Yaskawa INFORM job: DEMO_ROOF_SIDE_0625_3PAINT_13.JBI

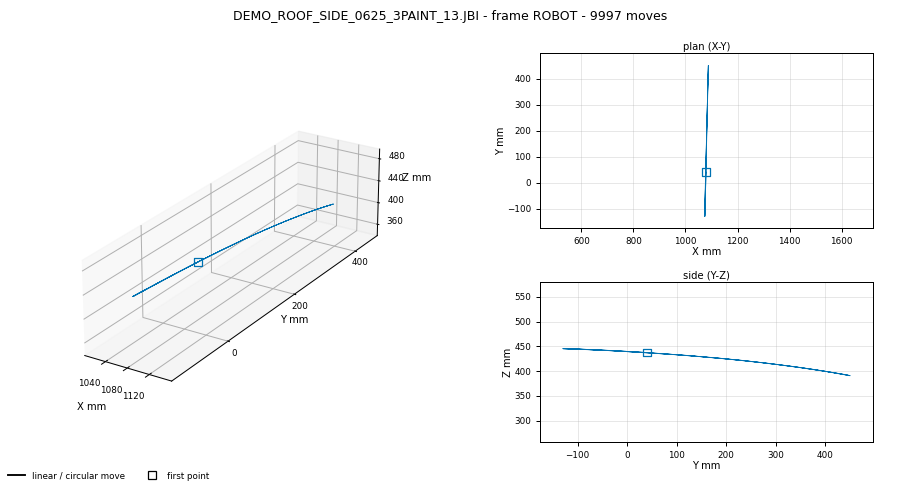
[picture p0: tool path of DEMO_ROOF_SIDE_0625_3PAINT_13.JBI in frame ROBOT, 9997 of 9997 moves have a stored position in this frame; points joined in program order, loops and branches not executed]
/JOB
//NAME DEMO_ROOF_SIDE_0625_3PAINT13
//POS
///NPOS 9997,0,0,0,0,0
///TOOL 0
///USER 0
///POSTYPE ROBOT
///RECTAN
///RCONF 1,0,0,0,0,0,0,0,0,0,0,0,0,0,0,0,0,0,0,0,0,0,0,0
C00000=1079.209,40.966,437.430,173.893,21.647,153.724
C00001=1079.203,40.716,437.445,173.891,21.644,153.724
C00002=1079.197,40.467,437.461,173.890,21.643,153.724
C00003=1079.192,40.217,437.477,173.889,21.640,153.724
C00004=1079.186,39.968,437.493,173.888,21.638,153.723
C00005=1079.181,39.718,437.508,173.885,21.635,153.723
C00006=1079.174,39.469,437.524,173.884,21.633,153.723
C00007=1079.169,39.220,437.539,173.883,21.630,153.723
C00008=1079.163,38.971,437.556,173.881,21.628,153.723
C00009=1079.157,38.721,437.571,173.880,21.625,153.722
C00010=1079.151,38.471,437.587,173.878,21.623,153.722
C00011=1079.145,38.222,437.602,173.877,21.621,153.722
C00012=1079.139,37.973,437.618,173.875,21.618,153.722
C00013=1079.134,37.723,437.634,173.874,21.616,153.721
C00014=1079.129,37.474,437.649,173.873,21.614,153.721
C00015=1079.122,37.225,437.665,173.870,21.611,153.721
C00016=1079.116,36.975,437.680,173.869,21.609,153.721
C00017=1079.111,36.725,437.696,173.868,21.606,153.720
C00018=1079.105,36.476,437.711,173.867,21.605,153.720
C00019=1079.099,36.226,437.726,173.865,21.602,153.720
C00020=1079.093,35.977,437.743,173.863,21.600,153.720
C00021=1079.087,35.727,437.758,173.862,21.597,153.719
C00022=1079.082,35.478,437.773,173.861,21.595,153.719
C00023=1079.076,35.229,437.789,173.859,21.592,153.719
C00024=1079.069,34.979,437.804,173.857,21.590,153.719
C00025=1079.064,34.729,437.820,173.856,21.588,153.719
C00026=1079.058,34.481,437.835,173.855,21.585,153.718
C00027=1079.052,34.231,437.850,173.853,21.583,153.718
C00028=1079.046,33.981,437.866,173.852,21.581,153.718
C00029=1079.041,33.732,437.881,173.850,21.578,153.718
C00030=1079.035,33.483,437.897,173.848,21.576,153.717
C00031=1079.029,33.233,437.912,173.847,21.573,153.717
C00032=1079.023,32.984,437.927,173.846,21.571,153.717
C00033=1079.017,32.734,437.943,173.845,21.569,153.717
C00034=1079.011,32.485,437.958,173.843,21.566,153.716
C00035=1079.006,32.235,437.973,173.841,21.564,153.716
C00036=1079.000,31.985,437.989,173.840,21.562,153.716
C00037=1078.994,31.736,438.004,173.839,21.559,153.716
C00038=1078.988,31.487,438.020,173.837,21.557,153.715
C00039=1078.982,31.206,438.037,173.835,21.554,153.715
C00040=1078.975,30.926,438.054,173.833,21.551,153.715
C00041=1078.969,30.646,438.071,173.832,21.549,153.715
C00042=1078.963,30.365,438.088,173.830,21.546,153.714
C00043=1078.956,30.116,438.104,173.829,21.544,153.714
C00044=1078.951,29.867,438.119,173.828,21.542,153.714
C00045=1078.945,29.617,438.134,173.826,21.539,153.714
C00046=1078.939,29.367,438.150,173.825,21.536,153.713
C00047=1078.933,29.118,438.164,173.823,21.534,153.713
C00048=1078.928,28.868,438.180,173.822,21.532,153.713
C00049=1078.923,28.619,438.195,173.820,21.529,153.713
C00050=1078.916,28.370,438.211,173.819,21.527,153.712
C00051=1078.909,28.120,438.225,173.818,21.524,153.712
C00052=1078.904,27.871,438.241,173.816,21.523,153.712
C00053=1078.898,27.622,438.256,173.814,21.520,153.712
C00054=1078.892,27.372,438.271,173.813,21.517,153.711
C00055=1078.887,27.123,438.286,173.812,21.515,153.711
C00056=1078.881,26.873,438.301,173.810,21.513,153.711
C00057=1078.875,26.624,438.316,173.808,21.510,153.711
C00058=1078.870,26.374,438.331,173.807,21.508,153.711
C00059=1078.863,26.124,438.346,173.806,21.506,153.710
C00060=1078.857,25.875,438.361,173.805,21.503,153.710
C00061=1078.852,25.625,438.376,173.803,21.501,153.710
C00062=1078.846,25.376,438.391,173.801,21.499,153.710
C00063=1078.840,25.126,438.407,173.800,21.496,153.709
C00064=1078.834,24.877,438.421,173.799,21.494,153.709
C00065=1078.828,24.628,438.436,173.798,21.492,153.709
C00066=1078.822,24.378,438.452,173.796,21.489,153.709
C00067=1078.817,24.129,438.466,173.794,21.487,153.708
C00068=1078.810,23.879,438.481,173.793,21.484,153.708
C00069=1078.805,23.630,438.496,173.792,21.482,153.708
C00070=1078.799,23.380,438.511,173.790,21.480,153.708
C00071=1078.794,23.131,438.526,173.789,21.477,153.707
C00072=1078.787,22.881,438.541,173.787,21.475,153.707
C00073=1078.781,22.631,438.556,173.786,21.473,153.707
C00074=1078.776,22.382,438.572,173.784,21.470,153.707
C00075=1078.770,22.133,438.586,173.783,21.468,153.707
C00076=1078.764,21.884,438.601,173.781,21.465,153.706
C00077=1078.758,21.634,438.617,173.780,21.463,153.706
C00078=1078.752,21.385,438.631,173.778,21.460,153.706
C00079=1078.746,21.135,438.646,173.777,21.458,153.706
C00080=1078.741,20.885,438.661,173.776,21.456,153.705
C00081=1078.735,20.635,438.675,173.774,21.454,153.705
C00082=1078.729,20.387,438.690,173.772,21.451,153.705
C00083=1078.724,20.137,438.706,173.771,21.449,153.705
C00084=1078.718,19.888,438.720,173.770,21.447,153.704
C00085=1078.711,19.638,438.735,173.769,21.444,153.704
C00086=1078.706,19.389,438.750,173.767,21.442,153.704
C00087=1078.700,19.138,438.765,173.765,21.439,153.704
C00088=1078.694,18.889,438.779,173.764,21.437,153.703
C00089=1078.688,18.640,438.794,173.763,21.435,153.703
C00090=1078.682,18.391,438.809,173.762,21.432,153.703
C00091=1078.677,18.141,438.824,173.759,21.430,153.703
C00092=1078.671,17.891,438.838,173.758,21.428,153.703
C00093=1078.665,17.642,438.853,173.757,21.425,153.702
C00094=1078.659,17.393,438.868,173.756,21.423,153.702
C00095=1078.653,17.143,438.883,173.754,21.420,153.702
C00096=1078.648,16.894,438.898,173.752,21.418,153.702
C00097=1078.641,16.643,438.912,173.751,21.416,153.701
C00098=1078.636,16.395,438.927,173.750,21.414,153.701
C00099=1078.629,16.145,438.941,173.749,21.411,153.701
C00100=1078.624,15.895,438.955,173.747,21.408,153.701
C00101=1078.618,15.645,438.971,173.745,21.407,153.700
C00102=1078.612,15.396,438.985,173.744,21.404,153.700
C00103=1078.606,15.118,439.002,173.742,21.401,153.700
C00104=1078.599,14.838,439.018,173.741,21.399,153.700
C00105=1078.593,14.560,439.034,173.739,21.396,153.699
C00106=1078.586,14.281,439.051,173.738,21.394,153.699
C00107=1078.581,14.031,439.065,173.737,21.391,153.699
C00108=1078.574,13.781,439.080,173.734,21.389,153.699
C00109=1078.569,13.532,439.095,173.733,21.386,153.698
C00110=1078.562,13.282,439.109,173.732,21.384,153.698
C00111=1078.557,13.033,439.123,173.731,21.382,153.698
C00112=1078.550,12.784,439.138,173.729,21.380,153.698
C00113=1078.545,12.534,439.152,173.727,21.377,153.698
C00114=1078.539,12.285,439.167,173.726,21.375,153.697
C00115=1078.533,12.035,439.181,173.725,21.373,153.697
C00116=1078.527,11.786,439.196,173.723,21.371,153.697
C00117=1078.521,11.536,439.211,173.722,21.368,153.697
C00118=1078.515,11.287,439.224,173.720,21.366,153.696
C00119=1078.509,11.037,439.239,173.719,21.363,153.696
C00120=1078.503,10.787,439.253,173.718,21.361,153.696
C00121=1078.497,10.538,439.268,173.717,21.359,153.696
C00122=1078.491,10.289,439.283,173.714,21.357,153.696
C00123=1078.486,10.039,439.297,173.713,21.354,153.695
C00124=1078.479,9.789,439.312,173.712,21.352,153.695
C00125=1078.474,9.540,439.325,173.711,21.350,153.695
C00126=1078.467,9.291,439.340,173.709,21.348,153.695
C00127=1078.461,9.041,439.354,173.707,21.345,153.694
C00128=1078.456,8.792,439.368,173.706,21.343,153.694
C00129=1078.449,8.542,439.382,173.705,21.340,153.694
C00130=1078.444,8.293,439.397,173.703,21.338,153.694
C00131=1078.438,8.042,439.411,173.702,21.336,153.693
C00132=1078.432,7.794,439.426,173.700,21.333,153.693
C00133=1078.426,7.544,439.440,173.699,21.331,153.693
C00134=1078.420,7.294,439.455,173.698,21.329,153.693
C00135=1078.415,7.045,439.469,173.697,21.327,153.693
C00136=1078.409,6.796,439.483,173.694,21.324,153.692
C00137=1078.403,6.546,439.497,173.693,21.322,153.692
C00138=1078.397,6.296,439.511,173.692,21.319,153.692
C00139=1078.391,6.047,439.526,173.691,21.317,153.692
C00140=1078.385,5.797,439.540,173.690,21.315,153.691
C00141=1078.380,5.548,439.555,173.687,21.312,153.691
C00142=1078.373,5.298,439.568,173.686,21.310,153.691
C00143=1078.367,5.048,439.582,173.685,21.308,153.691
C00144=1078.361,4.799,439.597,173.684,21.305,153.691
C00145=1078.356,4.550,439.611,173.682,21.304,153.690
C00146=1078.350,4.300,439.625,173.680,21.301,153.690
C00147=1078.344,4.050,439.639,173.679,21.299,153.690
C00148=1078.339,3.801,439.653,173.678,21.296,153.690
C00149=1078.332,3.551,439.668,173.677,21.294,153.689
C00150=1078.327,3.302,439.682,173.675,21.292,153.689
C00151=1078.321,3.052,439.696,173.673,21.289,153.689
C00152=1078.314,2.803,439.710,173.672,21.287,153.689
C00153=1078.309,2.553,439.724,173.671,21.284,153.688
C00154=1078.303,2.304,439.738,173.670,21.282,153.688
C00155=1078.297,2.055,439.753,173.668,21.280,153.688
C00156=1078.291,1.804,439.767,173.666,21.277,153.688
C00157=1078.286,1.555,439.781,173.665,21.275,153.688
C00158=1078.280,1.305,439.795,173.664,21.273,153.687
C00159=1078.275,1.056,439.809,173.663,21.271,153.687
C00160=1078.268,0.806,439.823,173.661,21.269,153.687
C00161=1078.262,0.557,439.837,173.659,21.266,153.687
C00162=1078.257,0.308,439.851,173.658,21.264,153.687
C00163=1078.251,0.058,439.865,173.657,21.261,153.686
C00164=1078.245,-0.192,439.879,173.655,21.259,153.686
C00165=1078.240,-0.442,439.893,173.654,21.257,153.686
C00166=1078.233,-0.691,439.906,173.652,21.254,153.686
C00167=1078.227,-0.968,439.923,173.651,21.252,153.685
C00168=1078.221,-1.244,439.938,173.649,21.249,153.685
C00169=1078.214,-1.522,439.953,173.648,21.246,153.685
C00170=1078.207,-1.799,439.969,173.647,21.244,153.684
C00171=1078.202,-2.048,439.983,173.644,21.242,153.684
C00172=1078.196,-2.298,439.997,173.643,21.239,153.684
C00173=1078.191,-2.547,440.011,173.642,21.237,153.684
C00174=1078.185,-2.797,440.024,173.641,21.235,153.684
C00175=1078.178,-3.046,440.039,173.640,21.233,153.683
C00176=1078.173,-3.296,440.053,173.638,21.230,153.683
C00177=1078.167,-3.545,440.067,173.636,21.228,153.683
C00178=1078.161,-3.795,440.080,173.635,21.225,153.683
C00179=1078.156,-4.044,440.094,173.634,21.223,153.683
C00180=1078.149,-4.294,440.108,173.632,21.221,153.682
C00181=1078.143,-4.544,440.122,173.630,21.218,153.682
C00182=1078.138,-4.793,440.135,173.629,21.217,153.682
C00183=1078.132,-5.043,440.149,173.628,21.214,153.682
C00184=1078.125,-5.292,440.164,173.627,21.212,153.681
C00185=1078.119,-5.542,440.177,173.625,21.210,153.681
C00186=1078.114,-5.791,440.191,173.624,21.208,153.681
C00187=1078.108,-6.041,440.205,173.622,21.205,153.681
C00188=1078.101,-6.291,440.218,173.621,21.203,153.681
C00189=1078.096,-6.540,440.232,173.619,21.201,153.680
C00190=1078.090,-6.789,440.245,173.618,21.199,153.680
C00191=1078.084,-7.039,440.259,173.617,21.196,153.680
C00192=1078.078,-7.288,440.273,173.615,21.194,153.680
C00193=1078.072,-7.539,440.287,173.614,21.191,153.680
C00194=1078.066,-7.788,440.300,173.612,21.189,153.679
C00195=1078.060,-8.037,440.314,173.611,21.187,153.679
C00196=1078.055,-8.287,440.328,173.610,21.185,153.679
C00197=1078.049,-8.536,440.341,173.608,21.183,153.679
C00198=1078.043,-8.786,440.355,173.607,21.180,153.679
C00199=1078.036,-9.036,440.369,173.605,21.178,153.678
C00200=1078.031,-9.285,440.382,173.604,21.176,153.678
C00201=1078.025,-9.535,440.396,173.603,21.174,153.678
C00202=1078.019,-9.784,440.409,173.601,21.172,153.678
C00203=1078.013,-10.034,440.423,173.599,21.169,153.677
C00204=1078.007,-10.283,440.437,173.598,21.167,153.677
C00205=1078.001,-10.532,440.450,173.597,21.164,153.677
C00206=1077.995,-10.783,440.463,173.596,21.162,153.677
C00207=1077.989,-11.033,440.477,173.594,21.160,153.677
C00208=1077.984,-11.282,440.491,173.592,21.157,153.676
C00209=1077.977,-11.531,440.504,173.591,21.156,153.676
C00210=1077.972,-11.781,440.518,173.590,21.153,153.676
C00211=1077.966,-12.030,440.531,173.588,21.151,153.676
C00212=1077.960,-12.280,440.545,173.587,21.149,153.676
C00213=1077.954,-12.529,440.558,173.586,21.147,153.675
C00214=1077.949,-12.779,440.572,173.584,21.144,153.675
C00215=1077.943,-13.028,440.585,173.582,21.142,153.675
C00216=1077.937,-13.279,440.599,173.581,21.140,153.675
C00217=1077.930,-13.528,440.612,173.580,21.138,153.675
C00218=1077.925,-13.778,440.626,173.579,21.135,153.674
C00219=1077.919,-14.027,440.639,173.578,21.133,153.674
C00220=1077.913,-14.276,440.653,173.575,21.131,153.674
C00221=1077.907,-14.526,440.666,173.574,21.128,153.674
C00222=1077.902,-14.776,440.679,173.573,21.126,153.674
C00223=1077.896,-15.025,440.693,173.572,21.124,153.673
C00224=1077.890,-15.275,440.707,173.570,21.122,153.673
C00225=1077.884,-15.525,440.719,173.568,21.120,153.673
C00226=1077.878,-15.774,440.732,173.567,21.117,153.673
C00227=1077.873,-16.023,440.746,173.566,21.115,153.672
C00228=1077.866,-16.273,440.760,173.564,21.113,153.672
C00229=1077.860,-16.523,440.773,173.563,21.111,153.672
C00230=1077.854,-16.773,440.786,173.562,21.109,153.672
C00231=1077.847,-17.048,440.801,173.560,21.106,153.672
C00232=1077.841,-17.323,440.815,173.559,21.104,153.671
C00233=1077.835,-17.598,440.830,173.556,21.101,153.671
C00234=1077.827,-17.874,440.844,173.555,21.099,153.671
C00235=1077.822,-18.123,440.858,173.554,21.097,153.671
C00236=1077.816,-18.373,440.871,173.553,21.095,153.671
C00237=1077.810,-18.622,440.884,173.552,21.092,153.670
C00238=1077.804,-18.872,440.898,173.549,21.090,153.670
C00239=1077.798,-19.121,440.911,173.548,21.088,153.670
C00240=1077.792,-19.371,440.924,173.547,21.086,153.670
C00241=1077.786,-19.620,440.937,173.546,21.084,153.670
C00242=1077.780,-19.870,440.951,173.544,21.082,153.670
C00243=1077.775,-20.120,440.963,173.543,21.080,153.669
C00244=1077.768,-20.369,440.977,173.541,21.077,153.669
C00245=1077.762,-20.618,440.990,173.540,21.075,153.669
C00246=1077.757,-20.869,441.003,173.538,21.073,153.669
C00247=1077.751,-21.118,441.016,173.537,21.071,153.669
C00248=1077.745,-21.368,441.029,173.536,21.068,153.668
C00249=1077.739,-21.617,441.042,173.534,21.066,153.668
C00250=1077.733,-21.867,441.056,173.532,21.064,153.668
C00251=1077.727,-22.116,441.068,173.531,21.062,153.668
C00252=1077.721,-22.366,441.082,173.530,21.060,153.668
C00253=1077.715,-22.616,441.094,173.529,21.058,153.667
C00254=1077.710,-22.865,441.108,173.527,21.056,153.667
C00255=1077.704,-23.115,441.121,173.526,21.053,153.667
C00256=1077.697,-23.364,441.134,173.525,21.051,153.667
C00257=1077.691,-23.614,441.147,173.523,21.049,153.667
C00258=1077.685,-23.864,441.160,173.521,21.047,153.666
C00259=1077.680,-24.113,441.174,173.520,21.044,153.666
C00260=1077.674,-24.363,441.186,173.519,21.042,153.666
C00261=1077.668,-24.612,441.199,173.517,21.040,153.666
C00262=1077.662,-24.862,441.212,173.516,21.038,153.666
C00263=1077.656,-25.111,441.225,173.514,21.035,153.665
C00264=1077.650,-25.362,441.238,173.513,21.033,153.665
C00265=1077.644,-25.611,441.252,173.511,21.031,153.665
C00266=1077.639,-25.860,441.264,173.510,21.029,153.665
C00267=1077.633,-26.110,441.276,173.509,21.027,153.665
C00268=1077.627,-26.359,441.290,173.508,21.025,153.664
C00269=1077.622,-26.609,441.303,173.505,21.023,153.664
C00270=1077.615,-26.859,441.316,173.504,21.021,153.664
C00271=1077.610,-27.109,441.329,173.503,21.018,153.664
C00272=1077.603,-27.358,441.342,173.502,21.016,153.664
C00273=1077.597,-27.608,441.355,173.500,21.014,153.664
C00274=1077.591,-27.858,441.367,173.499,21.012,153.663
C00275=1077.585,-28.107,441.380,173.498,21.010,153.663
C00276=1077.579,-28.357,441.393,173.496,21.008,153.663
C00277=1077.573,-28.606,441.406,173.494,21.006,153.663
C00278=1077.567,-28.856,441.419,173.493,21.003,153.663
C00279=1077.561,-29.106,441.431,173.492,21.001,153.663
C00280=1077.555,-29.355,441.445,173.490,20.999,153.662
C00281=1077.549,-29.605,441.457,173.489,20.997,153.662
C00282=1077.543,-29.854,441.470,173.488,20.996,153.662
C00283=1077.538,-30.103,441.483,173.486,20.993,153.662
C00284=1077.532,-30.353,441.495,173.484,20.991,153.662
C00285=1077.526,-30.602,441.508,173.483,20.989,153.662
C00286=1077.520,-30.852,441.521,173.482,20.987,153.661
C00287=1077.514,-31.102,441.534,173.481,20.985,153.661
C00288=1077.508,-31.351,441.547,173.479,20.983,153.661
C00289=1077.502,-31.601,441.559,173.478,20.981,153.661
C00290=1077.495,-31.851,441.571,173.476,20.978,153.661
C00291=1077.489,-32.101,441.584,173.474,20.976,153.661
C00292=1077.483,-32.349,441.597,173.473,20.974,153.660
C00293=1077.478,-32.599,441.609,173.472,20.972,153.660
C00294=1077.472,-32.849,441.622,173.471,20.970,153.660
C00295=1077.465,-33.124,441.636,173.469,20.968,153.660
C00296=1077.459,-33.398,441.651,173.467,20.966,153.660
C00297=1077.453,-33.673,441.664,173.466,20.964,153.659
C00298=1077.446,-33.948,441.678,173.464,20.961,153.659
C00299=1077.440,-34.197,441.691,173.462,20.959,153.659
C00300=1077.434,-34.446,441.704,173.461,20.957,153.659
C00301=1077.428,-34.696,441.716,173.460,20.955,153.659
C00302=1077.422,-34.945,441.728,173.458,20.953,153.659
C00303=1077.416,-35.195,441.741,173.457,20.951,153.658
C00304=1077.410,-35.445,441.753,173.456,20.949,153.658
C00305=1077.403,-35.694,441.766,173.455,20.947,153.658
C00306=1077.398,-35.944,441.779,173.453,20.944,153.658
C00307=1077.392,-36.194,441.791,173.451,20.942,153.658
C00308=1077.386,-36.443,441.804,173.450,20.940,153.658
C00309=1077.380,-36.693,441.816,173.449,20.938,153.657
C00310=1077.375,-36.943,441.829,173.447,20.936,153.657
C00311=1077.369,-37.192,441.841,173.446,20.934,153.657
C00312=1077.363,-37.442,441.854,173.445,20.932,153.657
C00313=1077.356,-37.691,441.866,173.442,20.930,153.657
C00314=1077.350,-37.941,441.879,173.441,20.928,153.657
C00315=1077.345,-38.190,441.891,173.440,20.926,153.656
C00316=1077.339,-38.440,441.904,173.438,20.924,153.656
C00317=1077.333,-38.690,441.916,173.437,20.922,153.656
C00318=1077.327,-38.940,441.929,173.436,20.920,153.656
C00319=1077.321,-39.190,441.941,173.434,20.918,153.656
C00320=1077.315,-39.439,441.953,173.433,20.916,153.656
C00321=1077.310,-39.689,441.965,173.431,20.913,153.656
C00322=1077.303,-39.938,441.979,173.430,20.911,153.655
C00323=1077.297,-40.187,441.991,173.428,20.909,153.655
C00324=1077.291,-40.437,442.003,173.427,20.907,153.655
C00325=1077.286,-40.686,442.015,173.426,20.906,153.655
C00326=1077.279,-40.936,442.027,173.424,20.904,153.655
C00327=1077.273,-41.186,442.040,173.423,20.902,153.655
C00328=1077.267,-41.436,442.052,173.422,20.900,153.654
C00329=1077.260,-41.685,442.064,173.420,20.897,153.654
C00330=1077.255,-41.935,442.077,173.418,20.895,153.654
C00331=1077.249,-42.184,442.089,173.417,20.893,153.654
C00332=1077.243,-42.434,442.102,173.416,20.891,153.654
C00333=1077.237,-42.684,442.114,173.414,20.889,153.654
C00334=1077.231,-42.933,442.126,173.413,20.887,153.653
C00335=1077.225,-43.183,442.138,173.412,20.885,153.653
C00336=1077.219,-43.433,442.150,173.410,20.883,153.653
C00337=1077.213,-43.682,442.163,173.409,20.882,153.653
C00338=1077.208,-43.932,442.175,173.407,20.879,153.653
C00339=1077.201,-44.182,442.186,173.405,20.878,153.653
C00340=1077.195,-44.432,442.199,173.404,20.876,153.653
C00341=1077.189,-44.682,442.211,173.403,20.874,153.652
C00342=1077.183,-44.930,442.223,173.401,20.872,153.652
C00343=1077.177,-45.180,442.236,173.400,20.870,153.652
C00344=1077.172,-45.430,442.248,173.399,20.868,153.652
C00345=1077.165,-45.679,442.260,173.397,20.866,153.652
C00346=1077.160,-45.929,442.272,173.396,20.864,153.652
C00347=1077.154,-46.179,442.285,173.394,20.861,153.652
C00348=1077.147,-46.428,442.297,173.392,20.859,153.651
C00349=1077.142,-46.678,442.308,173.391,20.858,153.651
C00350=1077.135,-46.928,442.320,173.390,20.856,153.651
C00351=1077.129,-47.178,442.333,173.388,20.854,153.651
C00352=1077.124,-47.427,442.345,173.387,20.852,153.651
C00353=1077.118,-47.676,442.357,173.386,20.850,153.651
C00354=1077.112,-47.926,442.369,173.384,20.848,153.651
C00355=1077.107,-48.176,442.381,173.383,20.846,153.650
C00356=1077.100,-48.426,442.393,173.381,20.844,153.650
C00357=1077.094,-48.676,442.405,173.380,20.842,153.650
C00358=1077.088,-48.924,442.417,173.378,20.840,153.650
C00359=1077.081,-49.200,442.431,173.377,20.838,153.650
C00360=1077.075,-49.474,442.444,173.376,20.836,153.650
C00361=1077.069,-49.749,442.457,173.373,20.833,153.650
C00362=1077.062,-50.024,442.470,173.372,20.831,153.649
C00363=1077.056,-50.273,442.482,173.371,20.829,153.649
C00364=1077.051,-50.524,442.494,173.369,20.828,153.649
C00365=1077.044,-50.773,442.506,173.368,20.826,153.649
C00366=1077.039,-51.023,442.518,173.367,20.824,153.649
C00367=1077.032,-51.272,442.530,173.364,20.821,153.649
C00368=1077.026,-51.522,442.541,173.363,20.820,153.649
C00369=1077.020,-51.772,442.554,173.362,20.818,153.649
C00370=1077.014,-52.021,442.565,173.360,20.816,153.648
C00371=1077.007,-52.271,442.577,173.359,20.815,153.648
C00372=1077.001,-52.521,442.589,173.357,20.813,153.648
C00373=1076.995,-52.770,442.601,173.356,20.811,153.648
C00374=1076.989,-53.020,442.613,173.355,20.809,153.648
C00375=1076.983,-53.270,442.625,173.353,20.807,153.648
C00376=1076.977,-53.519,442.636,173.352,20.805,153.648
C00377=1076.970,-53.768,442.648,173.351,20.803,153.648
C00378=1076.965,-54.019,442.660,173.348,20.801,153.648
C00379=1076.959,-54.268,442.672,173.347,20.799,153.647
C00380=1076.952,-54.517,442.684,173.346,20.798,153.647
C00381=1076.946,-54.768,442.695,173.344,20.796,153.647
C00382=1076.940,-55.017,442.707,173.343,20.794,153.647
C00383=1076.934,-55.266,442.719,173.341,20.792,153.647
C00384=1076.928,-55.517,442.731,173.340,20.791,153.647
C00385=1076.922,-55.766,442.742,173.339,20.789,153.647
C00386=1076.916,-56.016,442.754,173.337,20.787,153.647
C00387=1076.910,-56.265,442.765,173.336,20.785,153.647
C00388=1076.904,-56.515,442.778,173.334,20.783,153.646
C00389=1076.898,-56.765,442.789,173.333,20.781,153.646
C00390=1076.891,-57.014,442.801,173.331,20.779,153.646
C00391=1076.886,-57.264,442.812,173.329,20.777,153.646
C00392=1076.879,-57.514,442.824,173.328,20.776,153.646
C00393=1076.873,-57.763,442.835,173.327,20.774,153.646
C00394=1076.867,-58.013,442.847,173.325,20.772,153.646
C00395=1076.862,-58.263,442.859,173.324,20.771,153.646
C00396=1076.855,-58.512,442.871,173.322,20.769,153.646
C00397=1076.849,-58.762,442.882,173.321,20.767,153.645
C00398=1076.843,-59.011,442.893,173.320,20.765,153.645
C00399=1076.837,-59.261,442.906,173.318,20.763,153.645
C00400=1076.831,-59.511,442.917,173.317,20.761,153.645
C00401=1076.825,-59.761,442.928,173.315,20.760,153.645
C00402=1076.819,-60.010,442.940,173.314,20.758,153.645
C00403=1076.813,-60.260,442.952,173.312,20.756,153.645
C00404=1076.807,-60.509,442.963,173.310,20.754,153.645
C00405=1076.801,-60.759,442.974,173.309,20.752,153.645
C00406=1076.795,-61.009,442.987,173.308,20.751,153.645
C00407=1076.789,-61.259,442.998,173.306,20.749,153.644
C00408=1076.782,-61.508,443.010,173.305,20.747,153.644
C00409=1076.777,-61.758,443.021,173.303,20.745,153.644
C00410=1076.770,-62.007,443.033,173.302,20.743,153.644
C00411=1076.765,-62.257,443.044,173.301,20.742,153.644
C00412=1076.759,-62.507,443.055,173.299,20.740,153.644
C00413=1076.753,-62.756,443.067,173.298,20.738,153.644
C00414=1076.746,-63.006,443.078,173.296,20.736,153.644
C00415=1076.741,-63.256,443.090,173.295,20.735,153.644
C00416=1076.735,-63.506,443.102,173.294,20.733,153.643
C00417=1076.729,-63.755,443.113,173.292,20.731,153.643
C00418=1076.722,-64.005,443.124,173.290,20.729,153.643
C00419=1076.717,-64.254,443.135,173.289,20.727,153.643
C00420=1076.711,-64.504,443.148,173.287,20.726,153.643
C00421=1076.705,-64.754,443.159,173.286,20.724,153.643
C00422=1076.699,-65.003,443.170,173.284,20.722,153.643
C00423=1076.692,-65.280,443.183,173.283,20.720,153.643
C00424=1076.686,-65.556,443.196,173.282,20.718,153.643
C00425=1076.678,-65.831,443.208,173.279,20.716,153.643
C00426=1076.672,-66.108,443.220,173.278,20.714,153.643
C00427=1076.666,-66.357,443.232,173.277,20.712,153.642
C00428=1076.661,-66.607,443.243,173.275,20.711,153.642
C00429=1076.655,-66.857,443.254,173.274,20.709,153.642
C00430=1076.649,-67.107,443.266,173.272,20.708,153.642
C00431=1076.643,-67.356,443.277,173.271,20.706,153.642
C00432=1076.636,-67.606,443.288,173.269,20.704,153.642
C00433=1076.630,-67.856,443.299,173.268,20.702,153.642
C00434=1076.625,-68.105,443.312,173.266,20.701,153.642
C00435=1076.619,-68.355,443.323,173.265,20.699,153.642
C00436=1076.613,-68.605,443.334,173.264,20.697,153.642
C00437=1076.607,-68.855,443.345,173.262,20.695,153.641
C00438=1076.601,-69.104,443.356,173.260,20.693,153.641
C00439=1076.595,-69.353,443.367,173.259,20.691,153.641
C00440=1076.589,-69.603,443.379,173.257,20.690,153.641
C00441=1076.584,-69.853,443.390,173.256,20.688,153.641
C00442=1076.577,-70.103,443.401,173.254,20.687,153.641
C00443=1076.571,-70.352,443.413,173.253,20.685,153.641
C00444=1076.566,-70.602,443.424,173.251,20.683,153.641
C00445=1076.559,-70.852,443.435,173.250,20.682,153.641
C00446=1076.553,-71.101,443.446,173.249,20.680,153.641
C00447=1076.548,-71.351,443.457,173.247,20.678,153.641
C00448=1076.542,-71.601,443.469,173.246,20.676,153.641
C00449=1076.536,-71.850,443.480,173.244,20.675,153.641
C00450=1076.530,-72.100,443.491,173.243,20.673,153.640
C00451=1076.524,-72.350,443.502,173.241,20.671,153.640
C00452=1076.518,-72.599,443.513,173.240,20.669,153.640
C00453=1076.512,-72.849,443.524,173.239,20.668,153.640
C00454=1076.506,-73.099,443.535,173.237,20.666,153.640
C00455=1076.500,-73.349,443.546,173.236,20.665,153.640
C00456=1076.495,-73.598,443.557,173.234,20.663,153.640
C00457=1076.488,-73.848,443.568,173.233,20.661,153.640
C00458=1076.483,-74.097,443.581,173.231,20.660,153.640
C00459=1076.477,-74.347,443.591,173.230,20.658,153.640
C00460=1076.470,-74.597,443.602,173.229,20.656,153.640
C00461=1076.464,-74.846,443.613,173.227,20.655,153.640
C00462=1076.458,-75.096,443.624,173.226,20.653,153.640
C00463=1076.452,-75.346,443.635,173.223,20.651,153.639
C00464=1076.447,-75.595,443.646,173.222,20.649,153.639
C00465=1076.440,-75.846,443.657,173.220,20.648,153.639
C00466=1076.435,-76.095,443.668,173.219,20.647,153.639
C00467=1076.429,-76.345,443.679,173.217,20.645,153.639
C00468=1076.422,-76.595,443.690,173.216,20.643,153.639
C00469=1076.416,-76.844,443.700,173.214,20.642,153.639
C00470=1076.410,-77.093,443.711,173.213,20.640,153.639
C00471=1076.404,-77.344,443.723,173.212,20.638,153.639
C00472=1076.398,-77.593,443.733,173.210,20.637,153.639
C00473=1076.392,-77.843,443.744,173.209,20.635,153.639
C00474=1076.386,-78.093,443.756,173.207,20.633,153.639
C00475=1076.380,-78.342,443.766,173.206,20.632,153.639
C00476=1076.375,-78.592,443.777,173.204,20.630,153.639
C00477=1076.368,-78.842,443.788,173.203,20.629,153.639
C00478=1076.362,-79.091,443.799,173.201,20.628,153.639
C00479=1076.356,-79.341,443.810,173.200,20.626,153.639
C00480=1076.350,-79.590,443.821,173.198,20.624,153.639
C00481=1076.344,-79.840,443.832,173.197,20.623,153.639
C00482=1076.338,-80.090,443.843,173.195,20.621,153.638
C00483=1076.332,-80.339,443.853,173.194,20.620,153.638
C00484=1076.325,-80.589,443.864,173.192,20.618,153.638
C00485=1076.320,-80.839,443.874,173.191,20.616,153.638
C00486=1076.313,-81.089,443.885,173.189,20.615,153.638
C00487=1076.306,-81.367,443.897,173.188,20.614,153.638
C00488=1076.299,-81.646,443.909,173.186,20.612,153.638
C00489=1076.293,-81.924,443.921,173.184,20.610,153.638
C00490=1076.286,-82.202,443.933,173.183,20.608,153.638
C00491=1076.280,-82.452,443.944,173.181,20.607,153.638
C00492=1076.273,-82.702,443.954,173.180,20.605,153.638
C00493=1076.267,-82.951,443.965,173.178,20.604,153.638
C00494=1076.262,-83.201,443.976,173.177,20.602,153.638
C00495=1076.255,-83.450,443.986,173.175,20.601,153.638
C00496=1076.249,-83.701,443.997,173.173,20.600,153.638
C00497=1076.243,-83.950,444.008,173.172,20.598,153.638
C00498=1076.237,-84.199,444.018,173.170,20.597,153.638
C00499=1076.231,-84.450,444.029,173.169,20.595,153.638
C00500=1076.225,-84.699,444.040,173.167,20.594,153.638
C00501=1076.219,-84.949,444.050,173.166,20.592,153.638
C00502=1076.213,-85.198,444.061,173.164,20.591,153.638
C00503=1076.207,-85.449,444.072,173.163,20.589,153.638
C00504=1076.200,-85.698,444.082,173.161,20.588,153.638
C00505=1076.194,-85.947,444.093,173.160,20.587,153.638
C00506=1076.189,-86.197,444.103,173.158,20.585,153.638
C00507=1076.182,-86.447,444.114,173.157,20.584,153.638
C00508=1076.176,-86.697,444.125,173.155,20.582,153.638
C00509=1076.170,-86.946,444.135,173.154,20.581,153.638
C00510=1076.164,-87.196,444.145,173.152,20.579,153.638
C00511=1076.158,-87.446,444.156,173.151,20.578,153.638
C00512=1076.151,-87.695,444.167,173.149,20.576,153.638
C00513=1076.146,-87.945,444.178,173.148,20.575,153.638
C00514=1076.140,-88.195,444.187,173.146,20.574,153.638
C00515=1076.133,-88.445,444.198,173.145,20.572,153.638
C00516=1076.127,-88.694,444.209,173.143,20.571,153.638
C00517=1076.121,-88.944,444.219,173.141,20.569,153.638
C00518=1076.116,-89.194,444.230,173.140,20.568,153.637
C00519=1076.109,-89.443,444.240,173.138,20.566,153.637
C00520=1076.103,-89.694,444.251,173.137,20.565,153.637
C00521=1076.097,-89.943,444.261,173.135,20.563,153.637
C00522=1076.091,-90.192,444.272,173.134,20.562,153.637
C00523=1076.085,-90.442,444.282,173.132,20.561,153.637
C00524=1076.079,-90.692,444.292,173.131,20.559,153.637
C00525=1076.073,-90.941,444.303,173.129,20.558,153.637
C00526=1076.067,-91.192,444.314,173.129,20.557,153.637
C00527=1076.061,-91.441,444.324,173.127,20.555,153.637
C00528=1076.055,-91.691,444.334,173.126,20.554,153.637
C00529=1076.049,-91.940,444.344,173.124,20.553,153.637
C00530=1076.043,-92.190,444.355,173.122,20.551,153.637
C00531=1076.037,-92.440,444.365,173.121,20.550,153.637
C00532=1076.031,-92.689,444.376,173.119,20.548,153.637
C00533=1076.024,-92.940,444.386,173.118,20.547,153.637
C00534=1076.019,-93.189,444.396,173.116,20.546,153.637
C00535=1076.013,-93.439,444.407,173.115,20.544,153.637
C00536=1076.007,-93.688,444.417,173.113,20.543,153.637
C00537=1076.001,-93.938,444.428,173.112,20.541,153.637
C00538=1075.995,-94.188,444.437,173.110,20.540,153.637
C00539=1075.989,-94.437,444.448,173.108,20.539,153.637
C00540=1075.983,-94.687,444.458,173.107,20.537,153.637
C00541=1075.976,-94.937,444.469,173.105,20.536,153.637
C00542=1075.970,-95.187,444.479,173.104,20.535,153.637
C00543=1075.965,-95.436,444.489,173.102,20.533,153.637
C00544=1075.958,-95.686,444.499,173.101,20.532,153.637
C00545=1075.953,-95.936,444.510,173.099,20.531,153.637
C00546=1075.946,-96.186,444.519,173.098,20.529,153.637
C00547=1075.941,-96.435,444.530,173.096,20.528,153.637
C00548=1075.935,-96.685,444.540,173.095,20.526,153.637
C00549=1075.929,-96.934,444.551,173.093,20.525,153.637
C00550=1075.923,-97.184,444.560,173.091,20.524,153.637
C00551=1075.916,-97.465,444.572,173.090,20.522,153.637
C00552=1075.909,-97.746,444.583,173.088,20.521,153.637
C00553=1075.903,-98.026,444.595,173.087,20.520,153.637
C00554=1075.896,-98.307,444.607,173.085,20.518,153.637
C00555=1075.890,-98.556,444.616,173.084,20.517,153.637
C00556=1075.882,-98.806,444.627,173.082,20.516,153.637
C00557=1075.877,-99.056,444.637,173.080,20.514,153.637
C00558=1075.871,-99.306,444.647,173.079,20.513,153.637
C00559=1075.864,-99.555,444.657,173.077,20.512,153.637
C00560=1075.859,-99.805,444.667,173.076,20.511,153.637
C00561=1075.852,-100.055,444.677,173.074,20.509,153.637
C00562=1075.846,-100.304,444.687,173.072,20.508,153.637
C00563=1075.841,-100.555,444.697,173.071,20.507,153.637
C00564=1075.834,-100.804,444.707,173.069,20.505,153.637
C00565=1075.828,-101.054,444.717,173.068,20.505,153.638
C00566=1075.822,-101.303,444.728,173.066,20.503,153.638
C00567=1075.816,-101.554,444.738,173.065,20.502,153.638
C00568=1075.810,-101.803,444.747,173.063,20.501,153.638
C00569=1075.803,-102.052,444.757,173.062,20.500,153.638
C00570=1075.798,-102.303,444.768,173.060,20.499,153.638
C00571=1075.791,-102.552,444.777,173.059,20.497,153.638
C00572=1075.785,-102.802,444.787,173.057,20.496,153.638
C00573=1075.780,-103.052,444.798,173.056,20.495,153.638
C00574=1075.773,-103.301,444.807,173.054,20.494,153.638
C00575=1075.767,-103.551,444.817,173.053,20.492,153.638
C00576=1075.761,-103.800,444.827,173.051,20.491,153.638
C00577=1075.755,-104.051,444.837,173.049,20.490,153.638
C00578=1075.749,-104.300,444.847,173.048,20.489,153.638
C00579=1075.743,-104.550,444.857,173.046,20.487,153.638
C00580=1075.736,-104.799,444.867,173.044,20.487,153.638
C00581=1075.731,-105.049,444.877,173.043,20.485,153.638
C00582=1075.725,-105.299,444.886,173.041,20.484,153.638
C00583=1075.718,-105.548,444.897,173.040,20.483,153.638
C00584=1075.712,-105.798,444.906,173.039,20.482,153.638
C00585=1075.707,-106.048,444.916,173.037,20.481,153.638
C00586=1075.701,-106.298,444.926,173.036,20.479,153.638
C00587=1075.694,-106.548,444.936,173.034,20.478,153.638
C00588=1075.688,-106.797,444.946,173.032,20.477,153.638
C00589=1075.682,-107.047,444.955,173.031,20.476,153.638
C00590=1075.676,-107.297,444.966,173.029,20.475,153.638
C00591=1075.670,-107.547,444.975,173.027,20.474,153.638
C00592=1075.664,-107.797,444.985,173.026,20.472,153.638
C00593=1075.658,-108.046,444.995,173.024,20.471,153.639
C00594=1075.651,-108.296,445.005,173.023,20.471,153.639
C00595=1075.645,-108.545,445.014,173.022,20.470,153.639
C00596=1075.639,-108.795,445.024,173.020,20.469,153.639
C00597=1075.633,-109.045,445.033,173.018,20.467,153.639
C00598=1075.627,-109.295,445.043,173.017,20.466,153.639
C00599=1075.621,-109.544,445.054,173.015,20.465,153.639
C00600=1075.615,-109.794,445.063,173.013,20.464,153.639
C00601=1075.609,-110.044,445.073,173.012,20.463,153.639
C00602=1075.602,-110.294,445.082,173.010,20.462,153.639
C00603=1075.596,-110.543,445.092,173.008,20.461,153.639
C00604=1075.590,-110.793,445.101,173.007,20.459,153.639
C00605=1075.584,-111.043,445.111,173.006,20.459,153.639
C00606=1075.578,-111.293,445.121,173.004,20.458,153.639
C00607=1075.572,-111.543,445.130,173.003,20.456,153.639
C00608=1075.565,-111.792,445.140,173.001,20.456,153.639
C00609=1075.559,-112.042,445.150,172.999,20.455,153.639
C00610=1075.553,-112.292,445.160,172.998,20.453,153.639
C00611=1075.548,-112.541,445.169,172.996,20.452,153.640
C00612=1075.542,-112.791,445.179,172.994,20.451,153.640
C00613=1075.536,-113.040,445.189,172.993,20.450,153.640
C00614=1075.529,-113.290,445.198,172.992,20.449,153.640
C00615=1075.523,-113.568,445.209,172.989,20.448,153.640
C00616=1075.516,-113.847,445.219,172.988,20.447,153.640
C00617=1075.508,-114.124,445.230,172.986,20.446,153.640
C00618=1075.502,-114.402,445.240,172.985,20.444,153.640
C00619=1075.496,-114.652,445.250,172.983,20.443,153.640
C00620=1075.490,-114.902,445.259,172.981,20.443,153.640
C00621=1075.484,-115.151,445.269,172.980,20.442,153.640
C00622=1075.478,-115.401,445.279,172.979,20.441,153.640
C00623=1075.471,-115.651,445.288,172.977,20.440,153.640
C00624=1075.465,-115.901,445.298,172.975,20.439,153.641
C00625=1075.459,-116.151,445.307,172.973,20.438,153.641
C00626=1075.453,-116.400,445.317,172.972,20.437,153.641
C00627=1075.447,-116.650,445.326,172.970,20.436,153.641
C00628=1075.441,-116.900,445.336,172.968,20.435,153.641
C00629=1075.434,-117.150,445.346,172.968,20.434,153.641
C00630=1075.429,-117.399,445.355,172.966,20.433,153.641
C00631=1075.423,-117.649,445.364,172.964,20.432,153.641
C00632=1075.417,-117.899,445.373,172.963,20.431,153.641
C00633=1075.410,-118.148,445.382,172.961,20.430,153.641
C00634=1075.404,-118.398,445.392,172.959,20.429,153.641
C00635=1075.397,-118.648,445.401,172.957,20.428,153.641
C00636=1075.391,-118.898,445.411,172.956,20.427,153.642
C00637=1075.385,-119.148,445.420,172.955,20.426,153.642
C00638=1075.380,-119.397,445.430,172.953,20.425,153.642
C00639=1075.373,-119.647,445.439,172.952,20.425,153.642
C00640=1075.367,-119.896,445.449,172.950,20.424,153.642
C00641=1075.361,-120.147,445.458,172.948,20.423,153.642
C00642=1075.354,-120.396,445.467,172.946,20.422,153.642
C00643=1075.348,-120.646,445.476,172.945,20.421,153.642
C00644=1075.342,-120.896,445.486,172.944,20.420,153.642
C00645=1075.337,-121.145,445.495,172.942,20.419,153.642
C00646=1075.330,-121.395,445.504,172.940,20.418,153.642
C00647=1075.324,-121.645,445.514,172.939,20.417,153.643
C00648=1075.318,-121.895,445.523,172.937,20.416,153.643
C00649=1075.311,-122.144,445.532,172.935,20.415,153.643
C00650=1075.305,-122.394,445.541,172.933,20.414,153.643
C00651=1075.300,-122.643,445.551,172.933,20.414,153.643
C00652=1075.293,-122.893,445.560,172.931,20.413,153.643
C00653=1075.288,-123.144,445.569,172.929,20.412,153.643
C00654=1075.281,-123.393,445.579,172.927,20.411,153.643
C00655=1075.275,-123.643,445.588,172.926,20.410,153.643
C00656=1075.268,-123.893,445.597,172.924,20.410,153.644
C00657=1075.263,-124.142,445.606,172.923,20.409,153.644
C00658=1075.257,-124.392,445.615,172.921,20.408,153.644
C00659=1075.251,-124.642,445.625,172.920,20.407,153.644
C00660=1075.244,-124.891,445.634,172.918,20.406,153.644
C00661=1075.238,-125.142,445.643,172.916,20.405,153.644
C00662=1075.232,-125.391,445.652,172.914,20.405,153.644
C00663=1075.226,-125.641,445.661,172.913,20.404,153.644
C00664=1075.219,-125.890,445.670,172.912,20.403,153.644
C00665=1075.213,-126.141,445.679,172.910,20.402,153.644
C00666=1075.207,-126.390,445.689,172.908,20.401,153.645
C00667=1075.202,-126.640,445.698,172.907,20.401,153.645
C00668=1075.195,-126.890,445.706,172.905,20.400,153.645
C00669=1075.189,-127.139,445.716,172.903,20.399,153.645
C00670=1075.183,-127.389,445.725,172.902,20.398,153.645
C00671=1075.177,-127.640,445.734,172.900,20.397,153.645
C00672=1075.171,-127.890,445.743,172.898,20.397,153.645
C00673=1075.166,-128.141,445.752,172.897,20.396,153.645
C00674=1075.163,-128.391,445.763,172.896,20.394,153.645
C00675=1075.163,-128.645,445.774,172.895,20.390,153.645
C00676=1075.166,-128.898,445.788,172.894,20.387,153.644
C00677=1075.170,-129.151,445.801,172.894,20.383,153.644
C00678=1075.178,-129.401,445.815,172.894,20.377,153.643
C00679=1074.783,-129.424,445.662,172.849,20.507,153.674
C00680=1074.776,-129.173,445.647,172.849,20.513,153.675
C00681=1074.771,-128.921,445.633,172.849,20.517,153.675
C00682=1074.768,-128.667,445.621,172.850,20.521,153.676
C00683=1074.768,-128.414,445.610,172.851,20.524,153.676
C00684=1074.770,-128.163,445.599,172.852,20.526,153.677
C00685=1074.775,-127.912,445.588,172.853,20.527,153.677
C00686=1074.781,-127.662,445.579,172.855,20.528,153.677
C00687=1074.788,-127.412,445.571,172.856,20.529,153.676
C00688=1074.794,-127.162,445.561,172.858,20.529,153.676
C00689=1074.800,-126.911,445.552,172.860,20.530,153.676
C00690=1074.806,-126.662,445.543,172.861,20.531,153.676
C00691=1074.812,-126.413,445.534,172.863,20.532,153.676
C00692=1074.818,-126.163,445.525,172.865,20.533,153.676
C00693=1074.824,-125.913,445.516,172.867,20.534,153.676
C00694=1074.831,-125.663,445.507,172.867,20.534,153.676
C00695=1074.837,-125.413,445.497,172.869,20.535,153.676
C00696=1074.843,-125.163,445.488,172.871,20.536,153.675
C00697=1074.849,-124.914,445.479,172.873,20.537,153.675
C00698=1074.856,-124.664,445.470,172.874,20.538,153.675
C00699=1074.862,-124.415,445.461,172.876,20.539,153.675
C00700=1074.868,-124.164,445.452,172.877,20.539,153.675
C00701=1074.874,-123.914,445.442,172.879,20.540,153.675
C00702=1074.879,-123.665,445.433,172.880,20.541,153.675
C00703=1074.886,-123.416,445.424,172.882,20.542,153.675
C00704=1074.892,-123.165,445.415,172.884,20.543,153.675
C00705=1074.898,-122.916,445.406,172.886,20.544,153.674
C00706=1074.904,-122.666,445.396,172.887,20.545,153.674
C00707=1074.911,-122.416,445.386,172.888,20.545,153.674
C00708=1074.916,-122.167,445.377,172.890,20.546,153.674
C00709=1074.923,-121.917,445.369,172.892,20.547,153.674
C00710=1074.929,-121.667,445.359,172.894,20.548,153.674
C00711=1074.935,-121.417,445.350,172.895,20.549,153.674
C00712=1074.941,-121.167,445.340,172.897,20.550,153.674
C00713=1074.948,-120.918,445.331,172.899,20.551,153.674
C00714=1074.953,-120.668,445.322,172.899,20.551,153.674
C00715=1074.959,-120.418,445.313,172.901,20.552,153.673
C00716=1074.965,-120.168,445.303,172.903,20.553,153.673
C00717=1074.972,-119.919,445.294,172.905,20.554,153.673
C00718=1074.978,-119.669,445.285,172.906,20.555,153.673
C00719=1074.984,-119.419,445.275,172.908,20.556,153.673
C00720=1074.991,-119.169,445.265,172.910,20.557,153.673
C00721=1074.996,-118.920,445.256,172.911,20.558,153.673
C00722=1075.002,-118.670,445.247,172.912,20.559,153.673
C00723=1075.008,-118.420,445.238,172.914,20.560,153.673
C00724=1075.014,-118.170,445.228,172.916,20.560,153.673
C00725=1075.020,-117.920,445.219,172.917,20.562,153.673
C00726=1075.027,-117.671,445.210,172.919,20.563,153.673
C00727=1075.034,-117.421,445.200,172.921,20.564,153.672
C00728=1075.040,-117.171,445.191,172.923,20.565,153.672
C00729=1075.046,-116.922,445.181,172.923,20.565,153.672
C00730=1075.051,-116.672,445.172,172.925,20.567,153.672
C00731=1075.058,-116.423,445.162,172.927,20.567,153.672
C00732=1075.064,-116.173,445.153,172.928,20.568,153.672
C00733=1075.070,-115.923,445.143,172.930,20.569,153.672
C00734=1075.076,-115.673,445.134,172.932,20.571,153.672
C00735=1075.082,-115.423,445.124,172.933,20.572,153.672
C00736=1075.089,-115.174,445.114,172.935,20.572,153.672
C00737=1075.095,-114.924,445.105,172.936,20.573,153.672
C00738=1075.101,-114.674,445.095,172.938,20.574,153.672
C00739=1075.107,-114.424,445.086,172.939,20.575,153.672
C00740=1075.114,-114.146,445.075,172.941,20.576,153.671
C00741=1075.120,-113.868,445.065,172.943,20.578,153.671
C00742=1075.127,-113.590,445.055,172.945,20.579,153.671
C00743=1075.134,-113.313,445.044,172.947,20.580,153.671
C00744=1075.140,-113.062,445.033,172.948,20.581,153.671
C00745=1075.146,-112.813,445.024,172.949,20.582,153.671
C00746=1075.152,-112.563,445.014,172.951,20.583,153.671
C00747=1075.158,-112.313,445.005,172.953,20.584,153.671
C00748=1075.164,-112.063,444.995,172.954,20.585,153.671
C00749=1075.171,-111.813,444.986,172.956,20.586,153.671
C00750=1075.177,-111.564,444.976,172.958,20.587,153.671
C00751=1075.183,-111.314,444.966,172.959,20.588,153.671
C00752=1075.189,-111.064,444.957,172.961,20.590,153.671
C00753=1075.195,-110.814,444.947,172.963,20.590,153.671
C00754=1075.201,-110.564,444.938,172.964,20.592,153.671
C00755=1075.208,-110.315,444.927,172.965,20.592,153.670
C00756=1075.214,-110.066,444.918,172.967,20.593,153.670
C00757=1075.219,-109.815,444.908,172.968,20.595,153.670
C00758=1075.226,-109.566,444.898,172.970,20.596,153.670
C00759=1075.232,-109.316,444.889,172.972,20.597,153.670
C00760=1075.238,-109.066,444.879,172.973,20.598,153.670
C00761=1075.244,-108.816,444.869,172.975,20.599,153.670
C00762=1075.251,-108.567,444.859,172.977,20.600,153.670
C00763=1075.257,-108.317,444.850,172.978,20.601,153.670
C00764=1075.263,-108.067,444.840,172.980,20.603,153.670
C00765=1075.269,-107.818,444.830,172.982,20.604,153.670
C00766=1075.275,-107.568,444.821,172.982,20.605,153.670
C00767=1075.281,-107.318,444.811,172.984,20.605,153.670
C00768=1075.287,-107.069,444.800,172.986,20.607,153.670
C00769=1075.293,-106.819,444.791,172.987,20.608,153.670
C00770=1075.300,-106.569,444.781,172.989,20.609,153.670
C00771=1075.306,-106.319,444.772,172.991,20.610,153.670
C00772=1075.311,-106.070,444.761,172.992,20.612,153.670
C00773=1075.318,-105.820,444.751,172.994,20.613,153.670
C00774=1075.324,-105.570,444.742,172.995,20.614,153.670
C00775=1075.330,-105.320,444.732,172.997,20.615,153.670
C00776=1075.335,-105.070,444.722,172.999,20.616,153.669
C00777=1075.342,-104.821,444.712,173.000,20.618,153.669
C00778=1075.348,-104.571,444.702,173.002,20.619,153.669
C00779=1075.354,-104.321,444.693,173.003,20.620,153.669
C00780=1075.360,-104.072,444.682,173.004,20.621,153.669
C00781=1075.366,-103.822,444.672,173.006,20.622,153.669
C00782=1075.372,-103.572,444.663,173.007,20.623,153.669
C00783=1075.379,-103.323,444.653,173.009,20.624,153.669
C00784=1075.384,-103.073,444.642,173.011,20.626,153.669
C00785=1075.390,-102.823,444.633,173.012,20.627,153.669
C00786=1075.397,-102.573,444.623,173.014,20.628,153.669
C00787=1075.402,-102.324,444.612,173.015,20.629,153.669
C00788=1075.408,-102.074,444.603,173.017,20.631,153.669
C00789=1075.415,-101.824,444.593,173.019,20.632,153.669
C00790=1075.421,-101.575,444.583,173.020,20.633,153.669
C00791=1075.427,-101.325,444.573,173.022,20.634,153.669
C00792=1075.433,-101.075,444.563,173.023,20.636,153.669
C00793=1075.439,-100.826,444.553,173.025,20.637,153.669
C00794=1075.445,-100.576,444.543,173.026,20.637,153.669
C00795=1075.452,-100.326,444.532,173.027,20.639,153.669
C00796=1075.458,-100.076,444.522,173.029,20.640,153.669
C00797=1075.463,-99.826,444.512,173.030,20.642,153.669
C00798=1075.470,-99.577,444.502,173.032,20.643,153.669
C00799=1075.476,-99.327,444.492,173.034,20.644,153.669
C00800=1075.482,-99.078,444.481,173.035,20.646,153.669
C00801=1075.488,-98.828,444.472,173.037,20.646,153.669
C00802=1075.494,-98.578,444.462,173.038,20.648,153.669
C00803=1075.500,-98.329,444.451,173.040,20.649,153.669
C00804=1075.507,-98.048,444.440,173.042,20.651,153.669
C00805=1075.514,-97.767,444.429,173.043,20.652,153.669
C00806=1075.521,-97.486,444.417,173.046,20.654,153.669
C00807=1075.528,-97.205,444.406,173.047,20.655,153.669
C00808=1075.534,-96.956,444.395,173.049,20.656,153.669
C00809=1075.540,-96.706,444.386,173.050,20.658,153.669
C00810=1075.545,-96.456,444.375,173.052,20.659,153.669
C00811=1075.552,-96.207,444.365,173.053,20.661,153.669
C00812=1075.557,-95.957,444.354,173.055,20.662,153.669
C00813=1075.563,-95.707,444.345,173.057,20.663,153.669
C00814=1075.569,-95.458,444.334,173.057,20.664,153.669
C00815=1075.575,-95.208,444.324,173.059,20.666,153.669
C00816=1075.582,-94.958,444.313,173.060,20.667,153.669
C00817=1075.588,-94.708,444.304,173.062,20.668,153.669
C00818=1075.594,-94.458,444.293,173.063,20.670,153.669
C00819=1075.600,-94.209,444.283,173.065,20.671,153.669
C00820=1075.606,-93.959,444.272,173.067,20.672,153.669
C00821=1075.612,-93.709,444.263,173.068,20.674,153.669
C00822=1075.617,-93.460,444.252,173.070,20.675,153.669
C00823=1075.624,-93.210,444.242,173.071,20.677,153.669
C00824=1075.629,-92.961,444.231,173.073,20.678,153.669
C00825=1075.636,-92.710,444.220,173.074,20.679,153.669
C00826=1075.642,-92.461,444.211,173.076,20.681,153.669
C00827=1075.648,-92.211,444.200,173.077,20.682,153.669
C00828=1075.654,-91.961,444.190,173.079,20.684,153.669
C00829=1075.660,-91.712,444.179,173.080,20.685,153.669
C00830=1075.666,-91.463,444.169,173.082,20.687,153.669
C00831=1075.672,-91.212,444.158,173.083,20.688,153.669
C00832=1075.678,-90.962,444.148,173.085,20.689,153.669
C00833=1075.684,-90.713,444.138,173.087,20.690,153.669
C00834=1075.690,-90.463,444.127,173.088,20.692,153.669
C00835=1075.696,-90.214,444.117,173.090,20.693,153.669
C00836=1075.702,-89.964,444.107,173.091,20.695,153.669
C00837=1075.709,-89.714,444.096,173.093,20.696,153.669
C00838=1075.714,-89.464,444.085,173.094,20.698,153.669
C00839=1075.720,-89.214,444.075,173.096,20.699,153.669
C00840=1075.726,-88.965,444.065,173.097,20.700,153.669
C00841=1075.732,-88.716,444.054,173.099,20.702,153.669
C00842=1075.739,-88.466,444.043,173.100,20.703,153.669
C00843=1075.745,-88.216,444.033,173.102,20.705,153.669
C00844=1075.750,-87.966,444.022,173.103,20.706,153.669
C00845=1075.757,-87.717,444.012,173.105,20.708,153.669
C00846=1075.762,-87.467,444.002,173.107,20.709,153.669
C00847=1075.769,-87.217,443.990,173.108,20.711,153.669
C00848=1075.775,-86.968,443.980,173.110,20.712,153.669
C00849=1075.781,-86.718,443.969,173.111,20.713,153.669
C00850=1075.787,-86.468,443.960,173.113,20.715,153.669
C00851=1075.793,-86.218,443.948,173.114,20.716,153.669
C00852=1075.799,-85.969,443.938,173.116,20.718,153.669
C00853=1075.806,-85.719,443.927,173.117,20.719,153.669
C00854=1075.811,-85.469,443.917,173.119,20.721,153.670
C00855=1075.817,-85.219,443.906,173.120,20.723,153.670
C00856=1075.824,-84.970,443.896,173.122,20.724,153.670
C00857=1075.830,-84.720,443.885,173.123,20.725,153.670
C00858=1075.837,-84.471,443.874,173.125,20.727,153.670
C00859=1075.842,-84.220,443.864,173.126,20.728,153.670
C00860=1075.848,-83.971,443.853,173.128,20.730,153.670
C00861=1075.854,-83.722,443.843,173.129,20.731,153.670
C00862=1075.861,-83.472,443.832,173.131,20.733,153.670
C00863=1075.866,-83.222,443.821,173.132,20.734,153.670
C00864=1075.873,-82.973,443.810,173.134,20.736,153.670
C00865=1075.879,-82.722,443.800,173.135,20.737,153.670
C00866=1075.885,-82.473,443.789,173.137,20.738,153.670
C00867=1075.891,-82.223,443.779,173.138,20.740,153.670
C00868=1075.898,-81.945,443.767,173.140,20.742,153.670
C00869=1075.905,-81.666,443.754,173.141,20.743,153.670
C00870=1075.912,-81.388,443.743,173.143,20.745,153.670
C00871=1075.919,-81.110,443.730,173.145,20.747,153.670
C00872=1075.924,-80.860,443.720,173.147,20.749,153.670
C00873=1075.931,-80.610,443.708,173.148,20.750,153.670
C00874=1075.937,-80.361,443.698,173.150,20.751,153.670
C00875=1075.943,-80.111,443.687,173.151,20.753,153.670
C00876=1075.949,-79.860,443.677,173.153,20.754,153.670
C00877=1075.955,-79.611,443.666,173.154,20.756,153.670
C00878=1075.961,-79.362,443.656,173.155,20.758,153.670
C00879=1075.968,-79.111,443.644,173.157,20.759,153.670
C00880=1075.973,-78.862,443.633,173.159,20.761,153.670
C00881=1075.979,-78.613,443.623,173.160,20.762,153.670
C00882=1075.985,-78.362,443.611,173.161,20.764,153.671
C00883=1075.991,-78.113,443.600,173.163,20.765,153.671
C00884=1075.997,-77.863,443.590,173.164,20.767,153.671
C00885=1076.003,-77.613,443.578,173.166,20.769,153.671
C00886=1076.010,-77.364,443.568,173.167,20.770,153.671
C00887=1076.015,-77.114,443.557,173.169,20.772,153.671
C00888=1076.022,-76.864,443.546,173.170,20.773,153.671
C00889=1076.027,-76.615,443.535,173.172,20.775,153.671
C00890=1076.033,-76.365,443.524,173.173,20.777,153.671
C00891=1076.040,-76.115,443.513,173.175,20.778,153.671
C00892=1076.045,-75.866,443.502,173.176,20.780,153.671
C00893=1076.051,-75.616,443.491,173.178,20.781,153.671
C00894=1076.057,-75.366,443.480,173.179,20.783,153.671
C00895=1076.063,-75.116,443.469,173.181,20.784,153.671
C00896=1076.070,-74.868,443.458,173.182,20.786,153.671
C00897=1076.076,-74.618,443.447,173.183,20.788,153.671
C00898=1076.082,-74.368,443.436,173.185,20.789,153.672
C00899=1076.088,-74.118,443.425,173.186,20.791,153.672
C00900=1076.094,-73.869,443.414,173.188,20.793,153.672
C00901=1076.100,-73.619,443.403,173.189,20.795,153.672
C00902=1076.106,-73.369,443.392,173.191,20.796,153.672
C00903=1076.111,-73.119,443.380,173.192,20.798,153.672
C00904=1076.117,-72.870,443.369,173.194,20.799,153.672
C00905=1076.123,-72.619,443.358,173.195,20.801,153.672
C00906=1076.129,-72.371,443.346,173.196,20.803,153.672
C00907=1076.135,-72.121,443.336,173.199,20.805,153.672
C00908=1076.141,-71.871,443.324,173.200,20.807,153.672
C00909=1076.147,-71.621,443.313,173.202,20.808,153.672
C00910=1076.153,-71.372,443.303,173.203,20.810,153.673
C00911=1076.159,-71.122,443.291,173.205,20.812,153.673
C00912=1076.164,-70.872,443.279,173.206,20.814,153.673
C00913=1076.170,-70.623,443.268,173.207,20.815,153.673
C00914=1076.177,-70.373,443.257,173.209,20.817,153.673
C00915=1076.182,-70.123,443.246,173.210,20.818,153.673
C00916=1076.188,-69.874,443.235,173.212,20.820,153.673
C00917=1076.195,-69.624,443.223,173.213,20.822,153.673
C00918=1076.200,-69.375,443.212,173.214,20.824,153.673
C00919=1076.206,-69.124,443.201,173.216,20.825,153.673
C00920=1076.212,-68.875,443.190,173.217,20.827,153.673
C00921=1076.217,-68.625,443.179,173.219,20.829,153.673
C00922=1076.224,-68.376,443.167,173.220,20.831,153.674
C00923=1076.230,-68.126,443.156,173.222,20.832,153.674
C00924=1076.236,-67.876,443.145,173.223,20.834,153.674
C00925=1076.241,-67.626,443.133,173.224,20.835,153.674
C00926=1076.248,-67.377,443.121,173.226,20.837,153.674
C00927=1076.254,-67.127,443.110,173.227,20.839,153.674
C00928=1076.259,-66.878,443.100,173.230,20.841,153.674
C00929=1076.266,-66.628,443.088,173.231,20.843,153.674
C00930=1076.272,-66.379,443.077,173.232,20.845,153.674
C00931=1076.277,-66.128,443.065,173.234,20.847,153.674
C00932=1076.285,-65.852,443.053,173.235,20.848,153.674
C00933=1076.291,-65.576,443.040,173.237,20.850,153.675
C00934=1076.297,-65.300,443.028,173.239,20.853,153.675
C00935=1076.304,-65.023,443.014,173.240,20.854,153.675
C00936=1076.310,-64.774,443.004,173.242,20.856,153.675
C00937=1076.317,-64.524,442.992,173.243,20.858,153.675
C00938=1076.322,-64.274,442.980,173.244,20.859,153.675
C00939=1076.328,-64.024,442.969,173.246,20.861,153.675
C00940=1076.334,-63.775,442.957,173.247,20.863,153.675
C00941=1076.340,-63.525,442.946,173.249,20.865,153.675
C00942=1076.346,-63.276,442.935,173.250,20.867,153.676
C00943=1076.352,-63.026,442.923,173.251,20.868,153.676
C00944=1076.358,-62.776,442.912,173.253,20.870,153.676
C00945=1076.364,-62.527,442.900,173.254,20.872,153.676
C00946=1076.370,-62.277,442.889,173.256,20.874,153.676
C00947=1076.376,-62.027,442.876,173.258,20.876,153.676
C00948=1076.382,-61.778,442.866,173.259,20.877,153.676
C00949=1076.388,-61.528,442.854,173.261,20.879,153.676
C00950=1076.394,-61.279,442.843,173.262,20.881,153.676
C00951=1076.401,-61.029,442.831,173.264,20.883,153.676
C00952=1076.406,-60.779,442.819,173.265,20.885,153.677
C00953=1076.412,-60.529,442.808,173.266,20.886,153.677
C00954=1076.418,-60.280,442.796,173.268,20.888,153.677
C00955=1076.424,-60.030,442.785,173.269,20.890,153.677
C00956=1076.430,-59.781,442.773,173.271,20.892,153.677
C00957=1076.436,-59.531,442.762,173.272,20.894,153.677
C00958=1076.443,-59.281,442.750,173.273,20.895,153.677
C00959=1076.448,-59.031,442.738,173.275,20.897,153.677
C00960=1076.454,-58.782,442.726,173.277,20.899,153.677
C00961=1076.460,-58.532,442.715,173.278,20.901,153.678
C00962=1076.467,-58.283,442.704,173.280,20.903,153.678
C00963=1076.472,-58.034,442.691,173.281,20.905,153.678
C00964=1076.478,-57.783,442.680,173.282,20.907,153.678
C00965=1076.485,-57.534,442.668,173.284,20.908,153.678
C00966=1076.491,-57.284,442.657,173.285,20.910,153.678
C00967=1076.497,-57.034,442.645,173.287,20.912,153.678
C00968=1076.502,-56.785,442.634,173.288,20.914,153.678
C00969=1076.509,-56.535,442.622,173.289,20.915,153.678
C00970=1076.515,-56.285,442.609,173.291,20.917,153.679
C00971=1076.521,-56.036,442.598,173.292,20.919,153.679
C00972=1076.527,-55.786,442.586,173.295,20.921,153.679
C00973=1076.533,-55.536,442.575,173.296,20.923,153.679
C00974=1076.539,-55.287,442.563,173.297,20.925,153.679
C00975=1076.546,-55.037,442.551,173.299,20.927,153.679
C00976=1076.552,-54.787,442.540,173.300,20.929,153.679
C00977=1076.557,-54.538,442.528,173.301,20.931,153.679
C00978=1076.564,-54.288,442.516,173.303,20.932,153.679
C00979=1076.570,-54.038,442.504,173.304,20.934,153.680
C00980=1076.576,-53.789,442.492,173.306,20.936,153.680
C00981=1076.582,-53.540,442.480,173.307,20.937,153.680
C00982=1076.589,-53.289,442.469,173.308,20.939,153.680
C00983=1076.594,-53.040,442.457,173.310,20.941,153.680
C00984=1076.601,-52.791,442.445,173.312,20.944,153.680
C00985=1076.607,-52.540,442.434,173.313,20.945,153.680
C00986=1076.612,-52.291,442.421,173.315,20.947,153.680
C00987=1076.619,-52.042,442.410,173.316,20.949,153.681
C00988=1076.625,-51.791,442.398,173.317,20.951,153.681
C00989=1076.631,-51.542,442.386,173.319,20.953,153.681
C00990=1076.637,-51.293,442.374,173.320,20.955,153.681
C00991=1076.644,-51.043,442.362,173.322,20.957,153.681
C00992=1076.649,-50.793,442.350,173.323,20.958,153.681
C00993=1076.655,-50.544,442.339,173.324,20.960,153.681
C00994=1076.661,-50.294,442.326,173.326,20.962,153.681
C00995=1076.668,-50.044,442.314,173.328,20.964,153.682
C00996=1076.674,-49.770,442.301,173.329,20.966,153.682
C00997=1076.681,-49.494,442.287,173.331,20.968,153.682
C00998=1076.687,-49.220,442.274,173.333,20.971,153.682
C00999=1076.693,-48.944,442.262,173.334,20.973,153.682
C01000=1076.700,-48.695,442.250,173.335,20.975,153.682
C01001=1076.706,-48.445,442.237,173.337,20.977,153.682
C01002=1076.711,-48.196,442.225,173.338,20.979,153.683
C01003=1076.717,-47.946,442.213,173.339,20.981,153.683
C01004=1076.723,-47.696,442.201,173.341,20.982,153.683
C01005=1076.728,-47.447,442.189,173.342,20.984,153.683
C01006=1076.735,-47.197,442.177,173.344,20.987,153.683
C01007=1076.741,-46.947,442.165,173.346,20.989,153.683
C01008=1076.747,-46.698,442.153,173.347,20.991,153.684
C01009=1076.753,-46.448,442.140,173.348,20.993,153.684
C01010=1076.759,-46.198,442.128,173.350,20.995,153.684
C01011=1076.765,-45.949,442.116,173.351,20.996,153.684
C01012=1076.771,-45.700,442.104,173.352,20.998,153.684
C01013=1076.776,-45.449,442.092,173.354,21.000,153.684
C01014=1076.783,-45.200,442.080,173.355,21.002,153.684
C01015=1076.788,-44.950,442.068,173.357,21.005,153.684
C01016=1076.794,-44.701,442.055,173.359,21.006,153.685
C01017=1076.801,-44.451,442.043,173.360,21.008,153.685
C01018=1076.807,-44.201,442.031,173.361,21.010,153.685
C01019=1076.812,-43.952,442.019,173.363,21.012,153.685
C01020=1076.819,-43.702,442.007,173.364,21.014,153.685
C01021=1076.825,-43.452,441.994,173.365,21.016,153.685
C01022=1076.831,-43.203,441.981,173.367,21.018,153.686
C01023=1076.837,-42.954,441.970,173.368,21.020,153.686
C01024=1076.843,-42.704,441.957,173.370,21.023,153.686
C01025=1076.848,-42.454,441.945,173.371,21.025,153.686
C01026=1076.855,-42.204,441.933,173.373,21.027,153.686
C01027=1076.860,-41.955,441.921,173.374,21.029,153.686
C01028=1076.866,-41.705,441.908,173.375,21.031,153.687
C01029=1076.873,-41.456,441.896,173.377,21.033,153.687
C01030=1076.879,-41.206,441.884,173.378,21.034,153.687
C01031=1076.885,-40.956,441.871,173.379,21.036,153.687
C01032=1076.890,-40.707,441.859,173.382,21.039,153.687
C01033=1076.897,-40.457,441.847,173.383,21.041,153.687
C01034=1076.903,-40.207,441.834,173.384,21.043,153.687
C01035=1076.909,-39.957,441.822,173.386,21.045,153.688
C01036=1076.915,-39.708,441.810,173.387,21.047,153.688
C01037=1076.920,-39.459,441.798,173.388,21.049,153.688
C01038=1076.926,-39.209,441.785,173.390,21.051,153.688
C01039=1076.932,-38.959,441.773,173.391,21.053,153.688
C01040=1076.939,-38.710,441.760,173.392,21.055,153.688
C01041=1076.945,-38.460,441.747,173.394,21.057,153.689
C01042=1076.950,-38.211,441.735,173.396,21.059,153.689
C01043=1076.956,-37.961,441.723,173.397,21.061,153.689
C01044=1076.962,-37.711,441.710,173.398,21.063,153.689
C01045=1076.968,-37.461,441.697,173.400,21.065,153.689
C01046=1076.974,-37.211,441.685,173.401,21.067,153.689
C01047=1076.979,-36.962,441.673,173.402,21.069,153.690
C01048=1076.986,-36.713,441.660,173.404,21.071,153.690
C01049=1076.992,-36.463,441.647,173.406,21.074,153.690
C01050=1076.998,-36.213,441.635,173.407,21.076,153.690
C01051=1077.004,-35.964,441.622,173.408,21.078,153.690
C01052=1077.009,-35.714,441.610,173.410,21.080,153.690
C01053=1077.015,-35.464,441.598,173.411,21.082,153.691
C01054=1077.021,-35.215,441.584,173.412,21.084,153.691
C01055=1077.027,-34.965,441.572,173.414,21.086,153.691
C01056=1077.033,-34.715,441.559,173.416,21.088,153.691
C01057=1077.039,-34.466,441.547,173.417,21.090,153.691
C01058=1077.045,-34.216,441.534,173.418,21.092,153.691
C01059=1077.051,-33.967,441.521,173.420,21.094,153.692
C01060=1077.057,-33.692,441.508,173.421,21.096,153.692
C01061=1077.064,-33.418,441.494,173.423,21.099,153.692
C01062=1077.071,-33.143,441.480,173.424,21.101,153.692
C01063=1077.077,-32.868,441.466,173.426,21.104,153.692
C01064=1077.083,-32.619,441.453,173.427,21.106,153.693
C01065=1077.089,-32.369,441.440,173.429,21.108,153.693
C01066=1077.095,-32.119,441.428,173.430,21.110,153.693
C01067=1077.101,-31.870,441.415,173.432,21.112,153.693
C01068=1077.107,-31.621,441.402,173.433,21.114,153.693
C01069=1077.113,-31.371,441.390,173.434,21.116,153.693
C01070=1077.119,-31.121,441.377,173.436,21.118,153.694
C01071=1077.125,-30.872,441.364,173.437,21.120,153.694
C01072=1077.131,-30.622,441.352,173.439,21.123,153.694
C01073=1077.137,-30.372,441.339,173.440,21.125,153.694
C01074=1077.143,-30.123,441.326,173.442,21.127,153.694
C01075=1077.149,-29.873,441.313,173.443,21.129,153.694
C01076=1077.155,-29.623,441.301,173.444,21.131,153.695
C01077=1077.161,-29.374,441.287,173.446,21.133,153.695
C01078=1077.167,-29.124,441.275,173.447,21.135,153.695
C01079=1077.173,-28.875,441.262,173.449,21.138,153.695
C01080=1077.179,-28.625,441.249,173.450,21.139,153.695
C01081=1077.184,-28.376,441.237,173.452,21.141,153.695
C01082=1077.190,-28.126,441.224,173.453,21.144,153.696
C01083=1077.196,-27.877,441.211,173.454,21.146,153.696
C01084=1077.203,-27.627,441.198,173.456,21.148,153.696
C01085=1077.208,-27.377,441.185,173.457,21.150,153.696
C01086=1077.215,-27.128,441.172,173.459,21.152,153.696
C01087=1077.221,-26.878,441.159,173.460,21.155,153.697
C01088=1077.226,-26.628,441.147,173.462,21.157,153.697
C01089=1077.233,-26.379,441.133,173.463,21.159,153.697
C01090=1077.239,-26.129,441.121,173.464,21.161,153.697
C01091=1077.244,-25.880,441.107,173.465,21.163,153.697
C01092=1077.250,-25.630,441.095,173.467,21.165,153.698
C01093=1077.256,-25.380,441.081,173.469,21.167,153.698
C01094=1077.262,-25.131,441.069,173.470,21.170,153.698
C01095=1077.268,-24.881,441.055,173.471,21.172,153.698
C01096=1077.273,-24.631,441.042,173.473,21.174,153.698
C01097=1077.280,-24.382,441.029,173.474,21.176,153.699
C01098=1077.286,-24.132,441.016,173.475,21.178,153.699
C01099=1077.292,-23.883,441.003,173.477,21.181,153.699
C01100=1077.297,-23.634,440.991,173.479,21.183,153.699
C01101=1077.303,-23.384,440.977,173.480,21.185,153.699
C01102=1077.309,-23.134,440.965,173.481,21.187,153.700
C01103=1077.315,-22.885,440.951,173.482,21.189,153.700
C01104=1077.321,-22.636,440.938,173.484,21.192,153.700
C01105=1077.326,-22.385,440.925,173.485,21.194,153.700
C01106=1077.332,-22.136,440.912,173.487,21.196,153.700
C01107=1077.338,-21.886,440.899,173.489,21.198,153.700
C01108=1077.344,-21.637,440.886,173.490,21.200,153.701
C01109=1077.350,-21.387,440.873,173.491,21.202,153.701
C01110=1077.356,-21.137,440.859,173.492,21.204,153.701
C01111=1077.362,-20.888,440.846,173.493,21.207,153.701
C01112=1077.368,-20.638,440.834,173.496,21.209,153.702
C01113=1077.374,-20.389,440.820,173.497,21.211,153.702
C01114=1077.380,-20.139,440.806,173.498,21.214,153.702
C01115=1077.386,-19.890,440.794,173.499,21.216,153.702
C01116=1077.392,-19.640,440.780,173.501,21.218,153.702
C01117=1077.398,-19.390,440.766,173.502,21.220,153.703
C01118=1077.404,-19.140,440.754,173.504,21.223,153.703
C01119=1077.410,-18.891,440.741,173.505,21.225,153.703
C01120=1077.416,-18.642,440.727,173.507,21.227,153.703
C01121=1077.421,-18.391,440.714,173.508,21.229,153.703
C01122=1077.428,-18.142,440.701,173.509,21.231,153.703
C01123=1077.434,-17.893,440.688,173.510,21.233,153.704
C01124=1077.440,-17.617,440.673,173.513,21.236,153.704
C01125=1077.447,-17.342,440.658,173.514,21.238,153.704
C01126=1077.453,-17.066,440.643,173.516,21.241,153.704
C01127=1077.460,-16.792,440.629,173.517,21.243,153.705
C01128=1077.465,-16.542,440.616,173.518,21.245,153.705
C01129=1077.472,-16.292,440.603,173.520,21.247,153.705
C01130=1077.478,-16.042,440.589,173.521,21.250,153.705
C01131=1077.484,-15.793,440.575,173.523,21.252,153.705
C01132=1077.490,-15.543,440.563,173.524,21.254,153.706
C01133=1077.496,-15.294,440.549,173.526,21.256,153.706
C01134=1077.501,-15.044,440.535,173.527,21.258,153.706
C01135=1077.508,-14.795,440.522,173.528,21.261,153.706
C01136=1077.514,-14.546,440.509,173.529,21.263,153.706
C01137=1077.519,-14.295,440.496,173.532,21.265,153.707
C01138=1077.525,-14.046,440.483,173.533,21.268,153.707
C01139=1077.531,-13.796,440.469,173.534,21.270,153.707
C01140=1077.537,-13.547,440.455,173.535,21.272,153.707
C01141=1077.542,-13.298,440.442,173.537,21.274,153.707
C01142=1077.549,-13.048,440.428,173.538,21.277,153.708
C01143=1077.554,-12.797,440.415,173.540,21.279,153.708
C01144=1077.561,-12.548,440.401,173.541,21.282,153.708
C01145=1077.566,-12.299,440.388,173.542,21.284,153.708
C01146=1077.572,-12.049,440.374,173.544,21.285,153.709
C01147=1077.578,-11.800,440.360,173.545,21.288,153.709
C01148=1077.584,-11.551,440.347,173.546,21.290,153.709
C01149=1077.589,-11.301,440.333,173.548,21.293,153.709
C01150=1077.596,-11.052,440.320,173.550,21.295,153.709
C01151=1077.601,-10.801,440.307,173.551,21.297,153.710
C01152=1077.608,-10.552,440.293,173.552,21.299,153.710
C01153=1077.613,-10.302,440.279,173.553,21.301,153.710
C01154=1077.619,-10.052,440.266,173.555,21.304,153.710
C01155=1077.625,-9.803,440.252,173.557,21.306,153.710
C01156=1077.630,-9.554,440.238,173.558,21.309,153.711
C01157=1077.636,-9.304,440.225,173.559,21.311,153.711
C01158=1077.643,-9.054,440.211,173.560,21.313,153.711
C01159=1077.649,-8.805,440.198,173.562,21.315,153.711
C01160=1077.654,-8.555,440.184,173.564,21.318,153.712
C01161=1077.660,-8.306,440.171,173.565,21.320,153.712
C01162=1077.666,-8.056,440.157,173.566,21.322,153.712
C01163=1077.672,-7.807,440.143,173.568,21.324,153.712
C01164=1077.678,-7.557,440.129,173.569,21.326,153.712
C01165=1077.684,-7.307,440.115,173.571,21.329,153.713
C01166=1077.690,-7.058,440.102,173.572,21.331,153.713
C01167=1077.695,-6.808,440.088,173.573,21.334,153.713
C01168=1077.702,-6.559,440.075,173.575,21.336,153.713
C01169=1077.708,-6.309,440.061,173.576,21.338,153.714
C01170=1077.714,-6.060,440.047,173.577,21.340,153.714
C01171=1077.719,-5.810,440.034,173.579,21.342,153.714
C01172=1077.725,-5.561,440.019,173.581,21.345,153.714
C01173=1077.732,-5.311,440.005,173.582,21.347,153.714
C01174=1077.737,-5.061,439.991,173.583,21.349,153.715
C01175=1077.744,-4.812,439.978,173.584,21.351,153.715
C01176=1077.749,-4.563,439.964,173.586,21.354,153.715
C01177=1077.756,-4.313,439.951,173.588,21.356,153.715
C01178=1077.761,-4.063,439.937,173.589,21.359,153.715
C01179=1077.767,-3.814,439.923,173.590,21.361,153.716
C01180=1077.773,-3.564,439.910,173.592,21.363,153.716
C01181=1077.780,-3.315,439.895,173.593,21.365,153.716
C01182=1077.785,-3.065,439.881,173.595,21.367,153.716
C01183=1077.790,-2.815,439.867,173.596,21.370,153.717
C01184=1077.797,-2.566,439.854,173.597,21.372,153.717
C01185=1077.802,-2.317,439.840,173.599,21.374,153.717
C01186=1077.808,-2.066,439.826,173.600,21.377,153.717
C01187=1077.814,-1.817,439.811,173.602,21.379,153.717
C01188=1077.820,-1.541,439.796,173.603,21.382,153.718
C01189=1077.826,-1.263,439.780,173.604,21.384,153.718
C01190=1077.833,-0.986,439.765,173.606,21.387,153.718
C01191=1077.840,-0.709,439.749,173.607,21.390,153.719
C01192=1077.845,-0.460,439.735,173.610,21.392,153.719
C01193=1077.851,-0.210,439.722,173.611,21.394,153.719
C01194=1077.857,0.039,439.708,173.612,21.397,153.719
C01195=1077.863,0.289,439.693,173.613,21.399,153.719
C01196=1077.869,0.539,439.679,173.614,21.401,153.720
C01197=1077.874,0.788,439.665,173.616,21.403,153.720
C01198=1077.880,1.038,439.651,173.618,21.406,153.720
C01199=1077.886,1.287,439.636,173.619,21.408,153.720
C01200=1077.892,1.537,439.623,173.620,21.411,153.721
C01201=1077.898,1.786,439.609,173.621,21.413,153.721
C01202=1077.903,2.035,439.595,173.623,21.415,153.721
C01203=1077.910,2.285,439.580,173.625,21.418,153.721
C01204=1077.915,2.535,439.567,173.626,21.420,153.722
C01205=1077.921,2.785,439.553,173.627,21.422,153.722
C01206=1077.927,3.034,439.538,173.629,21.424,153.722
C01207=1077.932,3.284,439.524,173.630,21.427,153.722
C01208=1077.939,3.532,439.510,173.632,21.430,153.723
C01209=1077.944,3.782,439.496,173.633,21.432,153.723
C01210=1077.950,4.032,439.482,173.634,21.434,153.723
C01211=1077.956,4.281,439.467,173.636,21.436,153.723
C01212=1077.962,4.531,439.453,173.637,21.439,153.723
C01213=1077.968,4.781,439.439,173.639,21.441,153.724
C01214=1077.974,5.030,439.425,173.640,21.444,153.724
C01215=1077.979,5.280,439.411,173.641,21.446,153.724
C01216=1077.985,5.529,439.396,173.643,21.448,153.724
C01217=1077.991,5.779,439.382,173.644,21.450,153.725
C01218=1077.996,6.028,439.368,173.646,21.453,153.725
C01219=1078.004,6.278,439.354,173.647,21.455,153.725
C01220=1078.009,6.527,439.340,173.649,21.457,153.725
C01221=1078.015,6.776,439.325,173.650,21.460,153.726
C01222=1078.021,7.027,439.311,173.651,21.462,153.726
C01223=1078.027,7.276,439.296,173.653,21.465,153.726
C01224=1078.033,7.526,439.282,173.654,21.467,153.726
C01225=1078.038,7.775,439.268,173.656,21.469,153.726
C01226=1078.044,8.024,439.254,173.657,21.472,153.727
C01227=1078.050,8.274,439.239,173.658,21.473,153.727
C01228=1078.056,8.524,439.225,173.660,21.476,153.727
C01229=1078.062,8.773,439.210,173.661,21.479,153.727
C01230=1078.068,9.023,439.196,173.663,21.481,153.728
C01231=1078.073,9.272,439.181,173.664,21.483,153.728
C01232=1078.080,9.522,439.167,173.666,21.486,153.728
C01233=1078.085,9.771,439.153,173.667,21.488,153.728
C01234=1078.091,10.021,439.138,173.668,21.490,153.728
C01235=1078.097,10.270,439.124,173.670,21.493,153.729
C01236=1078.103,10.520,439.110,173.671,21.495,153.729
C01237=1078.109,10.769,439.095,173.673,21.497,153.729
C01238=1078.115,11.018,439.080,173.674,21.500,153.729
C01239=1078.121,11.269,439.066,173.676,21.502,153.730
C01240=1078.127,11.518,439.052,173.677,21.504,153.730
C01241=1078.133,11.768,439.037,173.678,21.506,153.730
C01242=1078.139,12.017,439.023,173.680,21.509,153.730
C01243=1078.144,12.266,439.008,173.681,21.511,153.731
C01244=1078.150,12.516,438.994,173.683,21.514,153.731
C01245=1078.156,12.765,438.979,173.684,21.516,153.731
C01246=1078.163,13.015,438.965,173.685,21.518,153.731
C01247=1078.168,13.264,438.951,173.687,21.520,153.731
C01248=1078.174,13.514,438.936,173.688,21.523,153.732
C01249=1078.180,13.763,438.921,173.690,21.525,153.732
C01250=1078.186,14.013,438.907,173.691,21.527,153.732
C01251=1078.192,14.262,438.892,173.693,21.530,153.732
C01252=1078.199,14.541,438.876,173.694,21.533,153.733
C01253=1078.205,14.820,438.860,173.696,21.535,153.733
C01254=1078.212,15.099,438.843,173.698,21.538,153.733
C01255=1078.218,15.379,438.827,173.699,21.540,153.733
C01256=1078.224,15.628,438.812,173.701,21.543,153.734
C01257=1078.230,15.877,438.798,173.702,21.545,153.734
C01258=1078.237,16.127,438.783,173.703,21.547,153.734
C01259=1078.242,16.376,438.769,173.704,21.550,153.734
C01260=1078.248,16.626,438.753,173.706,21.553,153.735
C01261=1078.253,16.875,438.739,173.708,21.555,153.735
C01262=1078.260,17.125,438.724,173.709,21.557,153.735
C01263=1078.265,17.375,438.710,173.710,21.559,153.735
C01264=1078.271,17.625,438.694,173.711,21.562,153.736
C01265=1078.277,17.873,438.680,173.713,21.565,153.736
C01266=1078.283,18.123,438.665,173.715,21.566,153.736
C01267=1078.289,18.372,438.650,173.716,21.569,153.736
C01268=1078.295,18.622,438.636,173.717,21.571,153.737
C01269=1078.300,18.872,438.621,173.719,21.574,153.737
C01270=1078.306,19.121,438.606,173.721,21.576,153.737
C01271=1078.312,19.370,438.591,173.722,21.578,153.737
C01272=1078.319,19.620,438.576,173.723,21.581,153.738
C01273=1078.324,19.869,438.561,173.724,21.583,153.738
C01274=1078.330,20.119,438.547,173.726,21.586,153.738
C01275=1078.335,20.368,438.533,173.728,21.588,153.738
C01276=1078.342,20.618,438.518,173.729,21.590,153.739
C01277=1078.347,20.867,438.502,173.730,21.592,153.739
C01278=1078.353,21.117,438.487,173.732,21.595,153.739
C01279=1078.358,21.366,438.472,173.733,21.598,153.739
C01280=1078.365,21.616,438.457,173.735,21.600,153.739
C01281=1078.371,21.865,438.443,173.736,21.602,153.740
C01282=1078.376,22.115,438.427,173.738,21.605,153.740
C01283=1078.382,22.364,438.413,173.739,21.607,153.740
C01284=1078.388,22.613,438.398,173.740,21.610,153.740
C01285=1078.394,22.864,438.383,173.742,21.612,153.741
C01286=1078.399,23.113,438.368,173.743,21.614,153.741
C01287=1078.406,23.363,438.353,173.745,21.617,153.741
C01288=1078.411,23.612,438.338,173.746,21.619,153.741
C01289=1078.417,23.862,438.323,173.747,21.621,153.742
C01290=1078.422,24.111,438.308,173.749,21.624,153.742
C01291=1078.429,24.360,438.293,173.751,21.626,153.742
C01292=1078.434,24.609,438.278,173.752,21.629,153.742
C01293=1078.440,24.859,438.263,173.753,21.631,153.743
C01294=1078.446,25.109,438.248,173.755,21.633,153.743
C01295=1078.452,25.358,438.233,173.757,21.636,153.743
C01296=1078.458,25.608,438.218,173.758,21.638,153.743
C01297=1078.464,25.857,438.203,173.759,21.640,153.744
C01298=1078.469,26.107,438.188,173.760,21.643,153.744
C01299=1078.476,26.356,438.172,173.762,21.646,153.744
C01300=1078.482,26.605,438.158,173.764,21.648,153.744
C01301=1078.487,26.855,438.142,173.765,21.650,153.745
C01302=1078.494,27.105,438.127,173.766,21.652,153.745
C01303=1078.499,27.354,438.112,173.767,21.654,153.745
C01304=1078.505,27.603,438.097,173.769,21.657,153.745
C01305=1078.510,27.853,438.082,173.771,21.659,153.745
C01306=1078.517,28.102,438.067,173.772,21.662,153.746
C01307=1078.522,28.352,438.051,173.773,21.664,153.746
C01308=1078.528,28.601,438.037,173.775,21.667,153.746
C01309=1078.534,28.851,438.020,173.776,21.669,153.747
C01310=1078.540,29.100,438.005,173.778,21.672,153.747
C01311=1078.545,29.350,437.990,173.779,21.673,153.747
C01312=1078.552,29.599,437.975,173.781,21.676,153.747
C01313=1078.557,29.848,437.960,173.782,21.679,153.748
C01314=1078.563,30.098,437.945,173.784,21.681,153.748
C01315=1078.569,30.347,437.929,173.785,21.683,153.748
C01316=1078.575,30.628,437.912,173.787,21.686,153.748
C01317=1078.582,30.908,437.895,173.788,21.689,153.749
C01318=1078.588,31.189,437.877,173.790,21.692,153.749
C01319=1078.595,31.469,437.860,173.792,21.694,153.749
C01320=1078.600,31.719,437.845,173.793,21.697,153.749
C01321=1078.606,31.968,437.830,173.795,21.699,153.750
C01322=1078.612,32.218,437.814,173.796,21.701,153.750
C01323=1078.618,32.467,437.799,173.798,21.704,153.750
C01324=1078.624,32.717,437.784,173.799,21.706,153.750
C01325=1078.629,32.967,437.768,173.800,21.709,153.751
C01326=1078.635,33.215,437.753,173.801,21.711,153.751
C01327=1078.641,33.465,437.738,173.804,21.713,153.751
C01328=1078.648,33.714,437.723,173.805,21.716,153.751
C01329=1078.653,33.964,437.706,173.806,21.718,153.752
C01330=1078.659,34.213,437.691,173.807,21.720,153.752
C01331=1078.665,34.463,437.676,173.809,21.723,153.752
C01332=1078.671,34.713,437.661,173.811,21.726,153.752
C01333=1078.676,34.961,437.645,173.812,21.728,153.752
C01334=1078.682,35.211,437.630,173.813,21.730,153.753
C01335=1078.688,35.461,437.614,173.815,21.733,153.753
C01336=1078.694,35.710,437.598,173.817,21.735,153.753
C01337=1078.700,35.959,437.583,173.818,21.737,153.753
C01338=1078.706,36.209,437.567,173.819,21.740,153.754
C01339=1078.711,36.459,437.552,173.821,21.742,153.754
C01340=1078.717,36.708,437.537,173.822,21.745,153.754
C01341=1078.723,36.957,437.521,173.823,21.747,153.755
C01342=1078.729,37.207,437.505,173.825,21.749,153.755
C01343=1078.735,37.456,437.490,173.827,21.752,153.755
C01344=1078.741,37.706,437.474,173.828,21.754,153.755
C01345=1078.746,37.955,437.459,173.829,21.756,153.755
C01346=1078.753,38.204,437.443,173.831,21.759,153.756
C01347=1078.758,38.454,437.428,173.833,21.761,153.756
C01348=1078.764,38.703,437.412,173.834,21.764,153.756
C01349=1078.769,38.953,437.396,173.835,21.766,153.756
C01350=1078.775,39.202,437.380,173.837,21.769,153.757
C01351=1078.781,39.452,437.365,173.839,21.771,153.757
C01352=1078.787,39.700,437.349,173.840,21.773,153.757
C01353=1078.793,39.950,437.334,173.841,21.776,153.757
C01354=1078.799,40.200,437.317,173.843,21.778,153.758
C01355=1078.804,40.450,437.302,173.844,21.781,153.758
C01356=1078.810,40.698,437.286,173.846,21.783,153.758
C01357=1078.815,40.948,437.270,173.847,21.785,153.758
C01358=1078.822,41.197,437.255,173.849,21.788,153.759
C01359=1078.828,41.447,437.239,173.850,21.790,153.759
C01360=1078.833,41.696,437.223,173.852,21.792,153.759
C01361=1078.839,41.946,437.208,173.854,21.795,153.759
C01362=1078.845,42.195,437.192,173.855,21.798,153.760
C01363=1078.850,42.445,437.176,173.856,21.800,153.760
C01364=1078.856,42.695,437.160,173.857,21.802,153.760
C01365=1078.861,42.944,437.145,173.859,21.805,153.760
C01366=1078.868,43.193,437.129,173.861,21.807,153.761
C01367=1078.874,43.442,437.113,173.862,21.809,153.761
C01368=1078.879,43.692,437.097,173.864,21.812,153.761
C01369=1078.885,43.942,437.081,173.865,21.814,153.761
C01370=1078.890,44.191,437.066,173.866,21.817,153.762
C01371=1078.896,44.440,437.049,173.868,21.819,153.762
C01372=1078.902,44.690,437.033,173.870,21.822,153.762
C01373=1078.908,44.939,437.018,173.871,21.824,153.762
C01374=1078.914,45.189,437.001,173.872,21.826,153.763
C01375=1078.919,45.438,436.985,173.873,21.829,153.763
C01376=1078.924,45.688,436.969,173.875,21.832,153.763
C01377=1078.930,45.937,436.953,173.877,21.834,153.763
C01378=1078.936,46.186,436.937,173.878,21.836,153.764
C01379=1078.941,46.436,436.922,173.880,21.839,153.764
C01380=1078.949,46.717,436.904,173.881,21.841,153.764
C01381=1078.955,46.997,436.885,173.883,21.844,153.764
C01382=1078.961,47.277,436.867,173.884,21.847,153.765
C01383=1078.967,47.558,436.849,173.887,21.850,153.765
C01384=1078.973,47.806,436.833,173.888,21.852,153.765
C01385=1078.978,48.056,436.818,173.889,21.854,153.765
C01386=1078.984,48.306,436.801,173.891,21.857,153.766
C01387=1078.990,48.555,436.785,173.892,21.859,153.766
C01388=1078.996,48.804,436.769,173.894,21.862,153.766
C01389=1079.002,49.054,436.752,173.896,21.864,153.766
C01390=1079.007,49.304,436.736,173.897,21.867,153.767
C01391=1079.013,49.553,436.721,173.898,21.869,153.767
C01392=1079.018,49.802,436.704,173.900,21.871,153.767
C01393=1079.024,50.051,436.688,173.902,21.874,153.767
C01394=1079.030,50.301,436.672,173.903,21.876,153.768
C01395=1079.036,50.551,436.656,173.904,21.878,153.768
C01396=1079.042,50.800,436.640,173.906,21.881,153.768
C01397=1079.047,51.050,436.623,173.907,21.884,153.769
C01398=1079.053,51.299,436.607,173.909,21.886,153.769
C01399=1079.058,51.548,436.591,173.911,21.888,153.769
C01400=1079.064,51.797,436.575,173.912,21.891,153.769
C01401=1079.070,52.047,436.559,173.913,21.893,153.769
C01402=1079.076,52.296,436.543,173.915,21.896,153.770
C01403=1079.082,52.546,436.527,173.917,21.898,153.770
C01404=1079.087,52.795,436.510,173.918,21.900,153.770
C01405=1079.093,53.045,436.494,173.919,21.903,153.770
C01406=1079.099,53.294,436.477,173.921,21.905,153.771
C01407=1079.105,53.543,436.461,173.923,21.907,153.771
C01408=1079.111,53.793,436.445,173.924,21.910,153.771
C01409=1079.117,54.042,436.429,173.926,21.913,153.771
C01410=1079.122,54.292,436.412,173.927,21.915,153.772
C01411=1079.128,54.541,436.395,173.928,21.917,153.772
C01412=1079.134,54.790,436.379,173.931,21.919,153.772
C01413=1079.139,55.039,436.363,173.932,21.922,153.772
C01414=1079.145,55.288,436.347,173.933,21.924,153.773
C01415=1079.151,55.538,436.331,173.934,21.926,153.773
C01416=1079.157,55.787,436.314,173.936,21.929,153.773
C01417=1079.162,56.037,436.298,173.938,21.932,153.773
C01418=1079.168,56.286,436.281,173.939,21.934,153.774
C01419=1079.174,56.536,436.265,173.941,21.936,153.774
C01420=1079.180,56.785,436.249,173.942,21.938,153.774
C01421=1079.186,57.035,436.232,173.944,21.941,153.774
C01422=1079.192,57.284,436.216,173.946,21.944,153.774
C01423=1079.197,57.533,436.200,173.947,21.946,153.775
C01424=1079.203,57.783,436.183,173.948,21.948,153.775
C01425=1079.209,58.032,436.166,173.950,21.950,153.775
C01426=1079.215,58.282,436.150,173.952,21.953,153.775
C01427=1079.221,58.531,436.134,173.953,21.955,153.776
C01428=1079.227,58.781,436.117,173.955,21.958,153.776
C01429=1079.233,59.030,436.101,173.956,21.960,153.776
C01430=1079.238,59.280,436.084,173.958,21.962,153.776
C01431=1079.244,59.529,436.068,173.959,21.964,153.777
C01432=1079.250,59.778,436.051,173.961,21.967,153.777
C01433=1079.256,60.027,436.035,173.962,21.969,153.777
C01434=1079.262,60.277,436.018,173.964,21.971,153.777
C01435=1079.268,60.526,436.002,173.966,21.974,153.777
C01436=1079.274,60.776,435.985,173.967,21.976,153.778
C01437=1079.279,61.025,435.969,173.968,21.978,153.778
C01438=1079.285,61.274,435.952,173.970,21.981,153.778
C01439=1079.291,61.524,435.935,173.972,21.983,153.778
C01440=1079.297,61.773,435.919,173.973,21.986,153.779
C01441=1079.303,62.022,435.903,173.975,21.988,153.779
C01442=1079.309,62.273,435.886,173.976,21.990,153.779
C01443=1079.315,62.521,435.869,173.978,21.992,153.779
C01444=1079.321,62.802,435.850,173.980,21.995,153.780
C01445=1079.328,63.081,435.832,173.982,21.998,153.780
C01446=1079.334,63.362,435.813,173.983,22.001,153.780
C01447=1079.341,63.642,435.794,173.985,22.003,153.780
C01448=1079.347,63.892,435.778,173.987,22.005,153.780
C01449=1079.353,64.141,435.761,173.988,22.007,153.781
C01450=1079.359,64.390,435.744,173.990,22.010,153.781
C01451=1079.364,64.639,435.728,173.991,22.013,153.781
C01452=1079.370,64.889,435.711,173.993,22.014,153.781
C01453=1079.376,65.138,435.694,173.995,22.017,153.782
C01454=1079.381,65.388,435.677,173.996,22.019,153.782
C01455=1079.388,65.638,435.660,173.997,22.022,153.782
C01456=1079.393,65.887,435.643,173.999,22.025,153.782
C01457=1079.399,66.136,435.626,174.001,22.027,153.783
C01458=1079.404,66.386,435.610,174.002,22.029,153.783
C01459=1079.411,66.634,435.593,174.004,22.031,153.783
C01460=1079.416,66.884,435.576,174.005,22.034,153.783
C01461=1079.422,67.133,435.560,174.007,22.036,153.783
C01462=1079.427,67.382,435.542,174.009,22.039,153.784
C01463=1079.433,67.632,435.526,174.010,22.041,153.784
C01464=1079.439,67.882,435.509,174.011,22.043,153.784
C01465=1079.445,68.131,435.492,174.013,22.046,153.784
C01466=1079.451,68.380,435.475,174.015,22.048,153.785
C01467=1079.457,68.629,435.458,174.016,22.050,153.785
C01468=1079.462,68.879,435.441,174.018,22.052,153.785
C01469=1079.468,69.128,435.424,174.019,22.055,153.785
C01470=1079.474,69.377,435.407,174.022,22.057,153.785
C01471=1079.480,69.627,435.390,174.023,22.060,153.786
C01472=1079.486,69.876,435.373,174.024,22.062,153.786
C01473=1079.491,70.126,435.356,174.026,22.064,153.786
C01474=1079.497,70.375,435.339,174.028,22.067,153.787
C01475=1079.502,70.624,435.322,174.029,22.069,153.787
C01476=1079.508,70.873,435.305,174.031,22.072,153.787
C01477=1079.514,71.123,435.288,174.032,22.074,153.787
C01478=1079.520,71.373,435.270,174.034,22.076,153.787
C01479=1079.525,71.622,435.254,174.036,22.079,153.788
C01480=1079.531,71.871,435.237,174.037,22.081,153.788
C01481=1079.537,72.121,435.220,174.038,22.083,153.788
C01482=1079.542,72.370,435.202,174.041,22.086,153.788
C01483=1079.549,72.620,435.186,174.042,22.088,153.789
C01484=1079.554,72.869,435.168,174.043,22.090,153.789
C01485=1079.560,73.118,435.150,174.045,22.093,153.789
C01486=1079.566,73.367,435.134,174.046,22.095,153.789
C01487=1079.571,73.616,435.117,174.049,22.098,153.789
C01488=1079.577,73.867,435.099,174.050,22.100,153.790
C01489=1079.582,74.116,435.082,174.051,22.102,153.790
C01490=1079.589,74.364,435.065,174.053,22.105,153.790
C01491=1079.594,74.614,435.048,174.055,22.107,153.790
C01492=1079.599,74.863,435.030,174.056,22.109,153.791
C01493=1079.606,75.113,435.014,174.058,22.112,153.791
C01494=1079.612,75.362,434.996,174.059,22.114,153.791
C01495=1079.617,75.611,434.979,174.061,22.116,153.791
C01496=1079.622,75.861,434.962,174.063,22.119,153.792
C01497=1079.629,76.110,434.944,174.064,22.121,153.792
C01498=1079.635,76.359,434.927,174.066,22.124,153.792
C01499=1079.640,76.609,434.910,174.068,22.125,153.792
C01500=1079.645,76.858,434.892,174.069,22.128,153.792
C01501=1079.652,77.107,434.875,174.071,22.130,153.793
C01502=1079.658,77.356,434.858,174.072,22.133,153.793
C01503=1079.663,77.606,434.841,174.074,22.135,153.793
C01504=1079.668,77.855,434.823,174.076,22.137,153.793
C01505=1079.675,78.105,434.805,174.077,22.139,153.793
C01506=1079.681,78.354,434.789,174.078,22.142,153.794
C01507=1079.686,78.603,434.771,174.081,22.144,153.794
C01508=1079.692,78.884,434.751,174.083,22.147,153.794
C01509=1079.699,79.163,434.732,174.084,22.149,153.794
C01510=1079.705,79.443,434.713,174.086,22.152,153.795
C01511=1079.712,79.724,434.692,174.088,22.155,153.795
C01512=1079.717,79.973,434.675,174.089,22.157,153.795
C01513=1079.723,80.222,434.657,174.091,22.159,153.795
C01514=1079.728,80.472,434.640,174.093,22.162,153.796
C01515=1079.734,80.722,434.623,174.094,22.164,153.796
C01516=1079.740,80.970,434.606,174.095,22.167,153.796
C01517=1079.746,81.219,434.588,174.098,22.169,153.796
C01518=1079.752,81.469,434.570,174.099,22.171,153.797
C01519=1079.757,81.718,434.553,174.101,22.174,153.797
C01520=1079.763,81.967,434.535,174.102,22.176,153.797
C01521=1079.768,82.217,434.518,174.104,22.178,153.797
C01522=1079.774,82.467,434.500,174.106,22.181,153.797
C01523=1079.780,82.716,434.483,174.107,22.183,153.798
C01524=1079.785,82.965,434.465,174.109,22.186,153.798
C01525=1079.791,83.214,434.447,174.111,22.188,153.798
C01526=1079.797,83.463,434.430,174.112,22.190,153.798
C01527=1079.802,83.712,434.412,174.114,22.192,153.798
C01528=1079.809,83.962,434.394,174.115,22.195,153.799
C01529=1079.814,84.211,434.376,174.117,22.197,153.799
C01530=1079.820,84.460,434.359,174.119,22.200,153.799
C01531=1079.826,84.710,434.341,174.120,22.202,153.799
C01532=1079.831,84.959,434.323,174.122,22.204,153.800
C01533=1079.837,85.208,434.306,174.124,22.206,153.800
C01534=1079.843,85.458,434.288,174.125,22.208,153.800
C01535=1079.848,85.707,434.270,174.127,22.211,153.800
C01536=1079.854,85.956,434.253,174.129,22.213,153.800
C01537=1079.860,86.206,434.235,174.131,22.216,153.801
C01538=1079.865,86.455,434.217,174.132,22.218,153.801
C01539=1079.872,86.704,434.199,174.133,22.220,153.801
C01540=1079.877,86.953,434.182,174.136,22.223,153.801
C01541=1079.883,87.203,434.164,174.137,22.224,153.801
C01542=1079.889,87.452,434.146,174.139,22.227,153.802
C01543=1079.894,87.702,434.128,174.140,22.229,153.802
C01544=1079.900,87.951,434.110,174.142,22.232,153.802
C01545=1079.905,88.200,434.093,174.144,22.234,153.802
C01546=1079.911,88.449,434.075,174.145,22.236,153.803
C01547=1079.917,88.699,434.057,174.147,22.239,153.803
C01548=1079.922,88.948,434.040,174.149,22.241,153.803
C01549=1079.928,89.198,434.022,174.150,22.243,153.803
C01550=1079.934,89.447,434.004,174.152,22.245,153.803
C01551=1079.940,89.696,433.985,174.154,22.247,153.804
C01552=1079.946,89.945,433.968,174.156,22.250,153.804
C01553=1079.951,90.194,433.950,174.157,22.252,153.804
C01554=1079.958,90.444,433.932,174.159,22.255,153.804
C01555=1079.963,90.693,433.915,174.161,22.257,153.804
C01556=1079.969,90.943,433.897,174.162,22.259,153.805
C01557=1079.974,91.191,433.878,174.164,22.262,153.805
C01558=1079.980,91.441,433.860,174.165,22.263,153.805
C01559=1079.986,91.690,433.842,174.168,22.266,153.805
C01560=1079.992,91.940,433.825,174.169,22.268,153.805
C01561=1079.997,92.189,433.806,174.170,22.271,153.806
C01562=1080.003,92.438,433.788,174.172,22.273,153.806
C01563=1080.009,92.687,433.770,174.174,22.275,153.806
C01564=1080.014,92.937,433.752,174.176,22.278,153.806
C01565=1080.020,93.187,433.734,174.177,22.280,153.806
C01566=1080.026,93.435,433.716,174.179,22.282,153.807
C01567=1080.032,93.685,433.698,174.181,22.284,153.807
C01568=1080.036,93.934,433.680,174.182,22.287,153.807
C01569=1080.042,94.183,433.662,174.184,22.289,153.807
C01570=1080.048,94.432,433.643,174.186,22.291,153.808
C01571=1080.053,94.682,433.625,174.188,22.294,153.808
C01572=1080.060,94.962,433.605,174.189,22.296,153.808
C01573=1080.067,95.242,433.585,174.191,22.299,153.808
C01574=1080.073,95.523,433.564,174.193,22.301,153.808
C01575=1080.079,95.802,433.544,174.196,22.304,153.809
C01576=1080.085,96.052,433.526,174.197,22.306,153.809
C01577=1080.090,96.301,433.507,174.199,22.309,153.809
C01578=1080.096,96.550,433.489,174.200,22.311,153.809
C01579=1080.102,96.799,433.472,174.202,22.313,153.810
C01580=1080.108,97.049,433.452,174.204,22.315,153.810
C01581=1080.113,97.298,433.435,174.205,22.318,153.810
C01582=1080.120,97.547,433.416,174.208,22.320,153.810
C01583=1080.124,97.796,433.398,174.209,22.322,153.810
C01584=1080.130,98.046,433.380,174.211,22.325,153.811
C01585=1080.136,98.295,433.362,174.212,22.327,153.811
C01586=1080.142,98.545,433.343,174.215,22.329,153.811
C01587=1080.148,98.794,433.325,174.216,22.331,153.811
C01588=1080.153,99.043,433.306,174.217,22.333,153.811
C01589=1080.159,99.292,433.288,174.220,22.336,153.811
C01590=1080.165,99.541,433.270,174.221,22.338,153.812
C01591=1080.171,99.791,433.251,174.223,22.340,153.812
C01592=1080.176,100.040,433.233,174.225,22.342,153.812
C01593=1080.182,100.289,433.215,174.227,22.345,153.812
C01594=1080.188,100.539,433.196,174.228,22.347,153.812
C01595=1080.194,100.787,433.178,174.230,22.349,153.813
C01596=1080.199,101.037,433.159,174.232,22.352,153.813
C01597=1080.205,101.286,433.141,174.233,22.354,153.813
C01598=1080.211,101.536,433.123,174.235,22.356,153.813
C01599=1080.217,101.785,433.104,174.236,22.358,153.814
C01600=1080.221,102.034,433.086,174.239,22.361,153.814
C01601=1080.228,102.283,433.067,174.240,22.363,153.814
C01602=1080.233,102.532,433.048,174.242,22.365,153.814
C01603=1080.239,102.782,433.030,174.244,22.367,153.814
C01604=1080.244,103.031,433.012,174.246,22.370,153.814
C01605=1080.250,103.280,432.994,174.247,22.372,153.815
C01606=1080.255,103.529,432.975,174.249,22.374,153.815
C01607=1080.261,103.779,432.955,174.251,22.376,153.815
C01608=1080.267,104.028,432.938,174.253,22.379,153.815
C01609=1080.272,104.277,432.919,174.254,22.381,153.815
C01610=1080.278,104.527,432.901,174.256,22.383,153.816
C01611=1080.284,104.776,432.882,174.258,22.386,153.816
C01612=1080.289,105.025,432.863,174.259,22.388,153.816
C01613=1080.295,105.275,432.845,174.262,22.390,153.816
C01614=1080.300,105.523,432.826,174.263,22.392,153.816
C01615=1080.307,105.773,432.807,174.265,22.395,153.817
C01616=1080.313,106.022,432.788,174.266,22.397,153.817
C01617=1080.317,106.271,432.770,174.269,22.399,153.817
C01618=1080.324,106.520,432.751,174.270,22.401,153.817
C01619=1080.329,106.769,432.732,174.272,22.404,153.817
C01620=1080.335,107.019,432.714,174.274,22.405,153.818
C01621=1080.341,107.268,432.695,174.276,22.408,153.818
C01622=1080.346,107.517,432.676,174.277,22.410,153.818
C01623=1080.352,107.766,432.658,174.279,22.413,153.818
C01624=1080.358,108.016,432.639,174.281,22.414,153.818
C01625=1080.363,108.265,432.620,174.283,22.417,153.819
C01626=1080.369,108.514,432.601,174.284,22.419,153.819
C01627=1080.375,108.764,432.582,174.287,22.421,153.819
C01628=1080.381,109.013,432.564,174.288,22.423,153.819
C01629=1080.386,109.262,432.545,174.290,22.426,153.819
C01630=1080.392,109.511,432.526,174.292,22.428,153.819
C01631=1080.398,109.761,432.508,174.294,22.430,153.820
C01632=1080.403,110.009,432.489,174.295,22.432,153.820
C01633=1080.409,110.259,432.469,174.297,22.435,153.820
C01634=1080.415,110.508,432.451,174.299,22.437,153.820
C01635=1080.421,110.757,432.431,174.301,22.439,153.820
C01636=1080.427,111.038,432.411,174.302,22.441,153.821
C01637=1080.433,111.318,432.389,174.305,22.444,153.821
C01638=1080.440,111.598,432.368,174.307,22.446,153.821
C01639=1080.446,111.878,432.347,174.309,22.449,153.821
C01640=1080.452,112.127,432.328,174.310,22.451,153.821
C01641=1080.457,112.376,432.309,174.313,22.453,153.821
C01642=1080.463,112.626,432.290,174.314,22.456,153.822
C01643=1080.469,112.875,432.271,174.316,22.458,153.822
C01644=1080.474,113.124,432.252,174.318,22.460,153.822
C01645=1080.480,113.373,432.233,174.320,22.462,153.822
C01646=1080.486,113.622,432.214,174.321,22.464,153.822
C01647=1080.492,113.872,432.195,174.323,22.467,153.823
C01648=1080.496,114.121,432.176,174.325,22.469,153.823
C01649=1080.502,114.371,432.157,174.327,22.471,153.823
C01650=1080.508,114.619,432.137,174.328,22.473,153.823
C01651=1080.514,114.869,432.118,174.331,22.476,153.823
C01652=1080.519,115.118,432.099,174.332,22.478,153.824
C01653=1080.525,115.367,432.080,174.334,22.480,153.824
C01654=1080.531,115.616,432.061,174.336,22.483,153.824
C01655=1080.537,115.866,432.042,174.338,22.485,153.824
C01656=1080.542,116.114,432.023,174.339,22.487,153.824
C01657=1080.547,116.364,432.004,174.342,22.489,153.824
C01658=1080.553,116.613,431.985,174.343,22.492,153.825
C01659=1080.558,116.862,431.966,174.345,22.494,153.825
C01660=1080.564,117.111,431.946,174.347,22.496,153.825
C01661=1080.569,117.361,431.927,174.349,22.498,153.825
C01662=1080.575,117.610,431.907,174.351,22.501,153.825
C01663=1080.580,117.859,431.888,174.352,22.503,153.826
C01664=1080.586,118.108,431.869,174.355,22.505,153.826
C01665=1080.591,118.357,431.849,174.356,22.507,153.826
C01666=1080.597,118.607,431.830,174.358,22.510,153.826
C01667=1080.603,118.856,431.811,174.359,22.512,153.826
C01668=1080.608,119.105,431.792,174.362,22.514,153.827
C01669=1080.614,119.354,431.773,174.363,22.516,153.827
C01670=1080.620,119.603,431.753,174.365,22.518,153.827
C01671=1080.625,119.853,431.733,174.367,22.521,153.827
C01672=1080.631,120.102,431.714,174.369,22.523,153.827
C01673=1080.636,120.351,431.695,174.370,22.525,153.827
C01674=1080.642,120.600,431.676,174.373,22.527,153.828
C01675=1080.648,120.849,431.656,174.375,22.529,153.828
C01676=1080.653,121.099,431.637,174.376,22.531,153.828
C01677=1080.659,121.348,431.618,174.379,22.534,153.828
C01678=1080.665,121.597,431.598,174.380,22.536,153.828
C01679=1080.670,121.846,431.579,174.382,22.538,153.828
C01680=1080.676,122.095,431.560,174.384,22.540,153.829
C01681=1080.681,122.345,431.540,174.386,22.543,153.829
C01682=1080.687,122.594,431.520,174.387,22.544,153.829
C01683=1080.692,122.843,431.501,174.389,22.547,153.829
C01684=1080.698,123.092,431.481,174.391,22.549,153.829
C01685=1080.704,123.341,431.461,174.393,22.551,153.830
C01686=1080.709,123.590,431.442,174.396,22.554,153.830
C01687=1080.715,123.839,431.423,174.397,22.556,153.830
C01688=1080.721,124.088,431.403,174.399,22.558,153.830
C01689=1080.727,124.338,431.384,174.401,22.560,153.830
C01690=1080.732,124.587,431.365,174.403,22.562,153.830
C01691=1080.738,124.836,431.344,174.404,22.564,153.830
C01692=1080.743,125.086,431.325,174.406,22.567,153.831
C01693=1080.749,125.335,431.306,174.408,22.569,153.831
C01694=1080.755,125.584,431.286,174.410,22.571,153.831
C01695=1080.761,125.833,431.267,174.412,22.573,153.831
C01696=1080.767,126.082,431.247,174.414,22.575,153.831
C01697=1080.772,126.332,431.227,174.416,22.578,153.831
C01698=1080.778,126.580,431.208,174.418,22.579,153.832
C01699=1080.783,126.829,431.188,174.420,22.582,153.832
C01700=1080.790,127.110,431.166,174.422,22.584,153.832
C01701=1080.796,127.390,431.144,174.424,22.587,153.832
C01702=1080.803,127.670,431.122,174.427,22.589,153.832
C01703=1080.809,127.950,431.100,174.428,22.591,153.832
C01704=1080.815,128.199,431.080,174.430,22.593,153.833
C01705=1080.821,128.449,431.060,174.433,22.596,153.833
C01706=1080.826,128.698,431.040,174.434,22.597,153.833
C01707=1080.832,128.947,431.021,174.436,22.600,153.833
C01708=1080.838,129.196,431.001,174.438,22.602,153.833
C01709=1080.843,129.445,430.981,174.440,22.604,153.833
C01710=1080.849,129.694,430.961,174.441,22.606,153.834
C01711=1080.855,129.944,430.942,174.444,22.608,153.834
C01712=1080.860,130.193,430.922,174.446,22.610,153.834
C01713=1080.866,130.441,430.902,174.448,22.612,153.834
C01714=1080.872,130.691,430.882,174.450,22.615,153.834
C01715=1080.878,130.940,430.862,174.451,22.617,153.834
C01716=1080.884,131.189,430.843,174.454,22.619,153.834
C01717=1080.889,131.438,430.823,174.456,22.621,153.835
C01718=1080.895,131.687,430.803,174.457,22.623,153.835
C01719=1080.900,131.937,430.783,174.460,22.625,153.835
C01720=1080.906,132.185,430.763,174.461,22.627,153.835
C01721=1080.912,132.434,430.743,174.463,22.629,153.835
C01722=1080.917,132.684,430.724,174.466,22.632,153.835
C01723=1080.923,132.933,430.703,174.467,22.634,153.836
C01724=1080.929,133.182,430.683,174.469,22.636,153.836
C01725=1080.934,133.431,430.664,174.471,22.638,153.836
C01726=1080.940,133.680,430.643,174.473,22.640,153.836
C01727=1080.946,133.929,430.623,174.475,22.642,153.836
C01728=1080.951,134.179,430.604,174.477,22.644,153.836
C01729=1080.957,134.428,430.584,174.479,22.647,153.836
C01730=1080.962,134.678,430.563,174.480,22.648,153.837
C01731=1080.968,134.926,430.543,174.483,22.651,153.837
C01732=1080.974,135.175,430.523,174.485,22.653,153.837
C01733=1080.979,135.425,430.503,174.487,22.655,153.837
C01734=1080.985,135.674,430.483,174.489,22.657,153.837
C01735=1080.991,135.923,430.462,174.491,22.660,153.837
C01736=1080.997,136.172,430.442,174.493,22.661,153.837
C01737=1081.002,136.421,430.423,174.495,22.664,153.838
C01738=1081.008,136.670,430.403,174.496,22.666,153.838
C01739=1081.013,136.919,430.382,174.499,22.668,153.838
C01740=1081.019,137.168,430.362,174.501,22.670,153.838
C01741=1081.024,137.417,430.342,174.502,22.672,153.838
C01742=1081.030,137.666,430.322,174.505,22.674,153.838
C01743=1081.036,137.916,430.301,174.507,22.677,153.838
C01744=1081.042,138.165,430.281,174.508,22.679,153.839
C01745=1081.047,138.415,430.261,174.511,22.681,153.839
C01746=1081.053,138.663,430.241,174.512,22.683,153.839
C01747=1081.058,138.912,430.220,174.514,22.685,153.839
C01748=1081.064,139.161,430.200,174.517,22.687,153.839
C01749=1081.069,139.410,430.180,174.518,22.689,153.839
C01750=1081.075,139.659,430.160,174.520,22.691,153.840
C01751=1081.081,139.908,430.139,174.523,22.694,153.840
C01752=1081.086,140.158,430.118,174.524,22.696,153.840
C01753=1081.092,140.407,430.098,174.526,22.698,153.840
C01754=1081.098,140.656,430.078,174.529,22.700,153.840
C01755=1081.104,140.905,430.058,174.530,22.702,153.840
C01756=1081.109,141.154,430.037,174.532,22.704,153.840
C01757=1081.114,141.403,430.017,174.534,22.706,153.841
C01758=1081.120,141.652,429.997,174.536,22.709,153.841
C01759=1081.125,141.901,429.976,174.539,22.711,153.841
C01760=1081.131,142.151,429.955,174.540,22.713,153.841
C01761=1081.137,142.400,429.935,174.542,22.715,153.841
C01762=1081.143,142.649,429.915,174.545,22.717,153.841
C01763=1081.148,142.898,429.894,174.546,22.719,153.842
C01764=1081.155,143.178,429.871,174.548,22.722,153.842
C01765=1081.160,143.458,429.849,174.551,22.724,153.842
C01766=1081.167,143.738,429.825,174.553,22.726,153.842
C01767=1081.173,144.018,429.802,174.555,22.728,153.842
C01768=1081.179,144.267,429.782,174.558,22.731,153.842
C01769=1081.185,144.517,429.761,174.560,22.733,153.842
C01770=1081.190,144.766,429.741,174.561,22.735,153.843
C01771=1081.195,145.015,429.720,174.564,22.737,153.843
C01772=1081.202,145.263,429.699,174.566,22.739,153.843
C01773=1081.207,145.513,429.678,174.567,22.741,153.843
C01774=1081.213,145.762,429.658,174.570,22.744,153.843
C01775=1081.219,146.011,429.638,174.572,22.746,153.843
C01776=1081.224,146.260,429.617,174.573,22.748,153.843
C01777=1081.229,146.509,429.597,174.576,22.750,153.843
C01778=1081.235,146.758,429.575,174.578,22.752,153.844
C01779=1081.241,147.007,429.555,174.580,22.754,153.844
C01780=1081.247,147.256,429.535,174.582,22.756,153.844
C01781=1081.252,147.505,429.514,174.584,22.758,153.844
C01782=1081.258,147.755,429.493,174.586,22.760,153.844
C01783=1081.264,148.003,429.473,174.588,22.762,153.844
C01784=1081.269,148.252,429.452,174.590,22.765,153.845
C01785=1081.274,148.502,429.431,174.593,22.766,153.845
C01786=1081.281,148.751,429.410,174.594,22.768,153.845
C01787=1081.286,149.000,429.389,174.597,22.771,153.845
C01788=1081.291,149.249,429.369,174.599,22.773,153.845
C01789=1081.297,149.498,429.347,174.600,22.775,153.845
C01790=1081.303,149.747,429.327,174.603,22.777,153.845
C01791=1081.309,149.996,429.307,174.605,22.779,153.845
C01792=1081.314,150.245,429.285,174.606,22.781,153.846
C01793=1081.320,150.495,429.264,174.609,22.784,153.846
C01794=1081.325,150.744,429.244,174.611,22.785,153.846
C01795=1081.331,150.992,429.223,174.613,22.788,153.846
C01796=1081.336,151.241,429.202,174.615,22.789,153.846
C01797=1081.342,151.490,429.180,174.617,22.792,153.846
C01798=1081.347,151.740,429.160,174.619,22.794,153.846
C01799=1081.353,151.989,429.139,174.621,22.796,153.847
C01800=1081.359,152.238,429.118,174.623,22.798,153.847
C01801=1081.364,152.487,429.097,174.626,22.800,153.847
C01802=1081.370,152.736,429.076,174.628,22.802,153.847
C01803=1081.375,152.985,429.055,174.629,22.804,153.847
C01804=1081.381,153.234,429.034,174.632,22.806,153.847
C01805=1081.386,153.483,429.013,174.634,22.809,153.847
C01806=1081.392,153.731,428.992,174.636,22.811,153.847
C01807=1081.398,153.981,428.971,174.638,22.813,153.848
C01808=1081.403,154.230,428.950,174.640,22.815,153.848
C01809=1081.409,154.480,428.929,174.643,22.817,153.848
C01810=1081.415,154.728,428.907,174.644,22.819,153.848
C01811=1081.420,154.977,428.887,174.646,22.821,153.848
C01812=1081.426,155.226,428.865,174.649,22.823,153.848
C01813=1081.431,155.476,428.845,174.650,22.825,153.848
C01814=1081.437,155.724,428.823,174.653,22.827,153.848
C01815=1081.443,155.974,428.802,174.655,22.829,153.848
C01816=1081.448,156.222,428.781,174.657,22.832,153.849
C01817=1081.454,156.471,428.760,174.659,22.833,153.849
C01818=1081.460,156.721,428.739,174.661,22.836,153.849
